LIN {X 0,Y 200.83,Z 502.645,A -85,B 0,C 180,E1 -22290.664,E2 -22290.664} C_VEL
LIN {X 0,Y 204.699,Z 493.667,A -85,B 0,C 180,E1 -22293.188,E2 -22293.188} C_VEL
LIN {X 0,Y 208.702,Z 483.459,A -85,B 0,C 180,E1 -22295.374,E2 -22295.374} C_VEL
LIN {X 0,Y 212.561,Z 471.698,A -85,B 0,C 180,E1 -22297.342,E2 -22297.342} C_VEL
LIN {X 0,Y 215.723,Z 459.835,A -85,B 0,C 180,E1 -22298.834,E2 -22298.834} C_VEL
LIN {X 0,Y 218.261,Z 447.534,A -85,B 0,C 180,E1 -22299.995,E2 -22299.995} C_VEL
LIN {X 0,Y 220.138,Z 434.92,A -85,B 0,C 180,E1 -22300.843,E2 -22300.843} C_VEL
LIN {X 0,Y 221.593,Z 419.626,A -85,B 0,C 180,E1 -22301.436,E2 -22301.436} C_VEL
LIN {X 0,Y 224.131,Z 384.01,A -85,B 0,C 180,E1 -22302.617,E2 -22302.617} C_VEL
LIN {X 0,Y 219.979,Z 374.841,A -85,B 0,C 180,E1 -22304.431,E2 -22304.431} C_VEL
LIN {X 0,Y 215.711,Z 367.271,A -85,B 0,C 180,E1 -22306.366,E2 -22306.366} C_VEL
LIN {X 0,Y 209.889,Z 358.051,A -85,B 0,C 180,E1 -22309.273,E2 -22309.273} C_VEL
LIN {X 0,Y 206.082,Z 352.787,A -85,B 0,C 180,E1 -22311.418,E2 -22311.418} C_VEL
LIN {X 0,Y 203.267,Z 348.749,A -85,B 0,C 180,E1 -22313.186,E2 -22313.186} C_VEL
LIN {X 0,Y 200.741,Z 345.417,A -85,B 0,C 180,E1 -22314.916,E2 -22314.916} C_VEL
LIN {X 0,Y 200.014,Z 344.287,A -85,B 0,C 180,E1 -22315.465,E2 -22315.465} C_VEL
LIN {X 0,Y 197.478,Z 341.831,A -85,B 0,C 180,E1 -22317.402,E2 -22317.402} C_VEL
LIN {X 0,Y 195.833,Z 338.802,A -85,B 0,C 180,E1 -22318.973,E2 -22318.973} C_VEL
LIN {X 0,Y 192.788,Z 336.052,A -85,B 0,C 180,E1 -22321.958,E2 -22321.958} C_VEL
LIN {X 0,Y 191.361,Z 333.353,A -85,B 0,C 180,E1 -22323.949,E2 -22323.949} C_VEL
LIN {X 0,Y 187.171,Z 330.783,A -85,B 0,C 180,E1 -22332.559,E2 -22332.559} C_VEL
LIN {X 0,Y 186.825,Z 330.456,A -85,B 0,C 180,E1 -22335.268,E2 -22335.268} C_VEL
LIN {X 0,Y 187.253,Z 331.063,A -85,B 0,C 180,E1 -22339.423,E2 -22339.423} C_VEL
LIN {X 0,Y 189.991,Z 333.324,A -85,B 0,C 180,E1 -22345.763,E2 -22345.763} C_VEL
LIN {X 0,Y 191.866,Z 335.584,A -85,B 0,C 180,E1 -22348.486,E2 -22348.486} C_VEL
LIN {X 0,Y 196.838,Z 342.088,A -85,B 0,C 180,E1 -22353.64,E2 -22353.64} C_VEL
LIN {X 0,Y 201.131,Z 348.366,A -85,B 0,C 180,E1 -22357.071,E2 -22357.071} C_VEL
LIN {X 0,Y 205.522,Z 355.246,A -85,B 0,C 180,E1 -22359.982,E2 -22359.982} C_VEL
LIN {X 0,Y 209.608,Z 362.229,A -85,B 0,C 180,E1 -22362.38,E2 -22362.38} C_VEL
LIN {X 0,Y 212.18,Z 366.87,A -85,B 0,C 180,E1 -22363.744,E2 -22363.744} C_VEL
LIN {X 0,Y 217.142,Z 376.724,A -85,B 0,C 180,E1 -22366.212,E2 -22366.212} C_VEL
LIN {X 0,Y 221.441,Z 387.148,A -85,B 0,C 180,E1 -22368.215,E2 -22368.215} C_VEL
LIN {X 0,Y 222.84,Z 391.134,A -85,B 0,C 180,E1 -22368.865,E2 -22368.865} C_VEL
LIN {X 0,Y 223.267,Z 398.392,A -85,B 0,C 180,E1 -22369.389,E2 -22369.389} C_VEL
LIN {X 0,Y 222.151,Z 414.024,A -85,B 0,C 180,E1 -22369.907,E2 -22369.907} C_VEL
LIN {X 0,Y 221.34,Z 419.86,A -85,B 0,C 180,E1 -22369.978,E2 -22369.978} C_VEL
LIN {X 0,Y 216.043,Z 438.883,A -85,B 0,C 180,E1 -22369.491,E2 -22369.491} C_VEL
LIN {X 0,Y 214.87,Z 444.674,A -85,B 0,C 180,E1 -22369.599,E2 -22369.599} C_VEL
LIN {X 0,Y 212.693,Z 457.533,A -85,B 0,C 180,E1 -22370.384,E2 -22370.384} C_VEL
LIN {X 0,Y 209.856,Z 469.525,A -85,B 0,C 180,E1 -22371.421,E2 -22371.421} C_VEL
LIN {X 0,Y 206.39,Z 481.375,A -85,B 0,C 180,E1 -22372.824,E2 -22372.824} C_VEL
LIN {X 0,Y 202.69,Z 492.094,A -85,B 0,C 180,E1 -22374.505,E2 -22374.505} C_VEL
LIN {X 0,Y 198.299,Z 502.866,A -85,B 0,C 180,E1 -22376.689,E2 -22376.689} C_VEL
LIN {X 0,Y 194.337,Z 511.664,A -85,B 0,C 180,E1 -22378.99,E2 -22378.99} C_VEL
LIN {X 0,Y 190.029,Z 520.315,A -85,B 0,C 180,E1 -22381.875,E2 -22381.875} C_VEL
LIN {X 0,Y 186.598,Z 526.823,A -85,B 0,C 180,E1 -22384.68,E2 -22384.68} C_VEL
LIN {X 0,Y 183.631,Z 532.054,A -85,B 0,C 180,E1 -22387.507,E2 -22387.507} C_VEL
LIN {X 0,Y 180.942,Z 536.694,A -85,B 0,C 180,E1 -22390.731,E2 -22390.731} C_VEL
LIN {X 0,Y 178.737,Z 540.277,A -85,B 0,C 180,E1 -22394.032,E2 -22394.032} C_VEL
LIN {X 0,Y 177.762,Z 542.118,A -85,B 0,C 180,E1 -22396.286,E2 -22396.286} C_VEL
LIN {X 0,Y 176.452,Z 544.563,A -85,B 0,C 180,E1 -22400.841,E2 -22400.841} C_VEL
LIN {X 0,Y 176.134,Z 545.21,A -85,B 0,C 180,E1 -22403.133,E2 -22403.133} C_VEL
LIN {X 0,Y 175.989,Z 545.399,A -85,B 0,C 180,E1 -22406.716,E2 -22406.716} C_VEL
LIN {X 0,Y 176.24,Z 544.71,A -85,B 0,C 180,E1 -22410.007,E2 -22410.007} C_VEL
LIN {X 0,Y 176.072,Z 542.876,A -85,B 0,C 180,E1 -22413.72,E2 -22413.72} C_VEL
LIN {X 0,Y 176.313,Z 539.323,A -85,B 0,C 180,E1 -22418.027,E2 -22418.027} C_VEL
LIN {X 0,Y 176.918,Z 535.242,A -85,B 0,C 180,E1 -22421.463,E2 -22421.463} C_VEL
LIN {X 0,Y 178.269,Z 528.927,A -85,B 0,C 180,E1 -22425.439,E2 -22425.439} C_VEL
LIN {X 0,Y 180.034,Z 522.023,A -85,B 0,C 180,E1 -22428.794,E2 -22428.794} C_VEL
LIN {X 0,Y 181.845,Z 515.368,A -85,B 0,C 180,E1 -22431.388,E2 -22431.388} C_VEL
LIN {X 0,Y 184.238,Z 506.448,A -85,B 0,C 180,E1 -22434.215,E2 -22434.215} C_VEL
LIN {X 0,Y 186.613,Z 497.088,A -85,B 0,C 180,E1 -22436.571,E2 -22436.571} C_VEL
LIN {X 0,Y 189.347,Z 485.491,A -85,B 0,C 180,E1 -22438.856,E2 -22438.856} C_VEL
LIN {X 0,Y 191.354,Z 475.884,A -85,B 0,C 180,E1 -22440.337,E2 -22440.337} C_VEL
LIN {X 0,Y 193.525,Z 463.742,A -85,B 0,C 180,E1 -22441.78,E2 -22441.78} C_VEL
LIN {X 0,Y 195.313,Z 450.462,A -85,B 0,C 180,E1 -22442.888,E2 -22442.888} C_VEL
LIN {X 0,Y 196.507,Z 437.019,A -85,B 0,C 180,E1 -22443.598,E2 -22443.598} C_VEL
LIN {X 0,Y 198.622,Z 393.171,A -85,B 0,C 180,E1 -22445.244,E2 -22445.244} C_VEL
LIN {X 0,Y 196.265,Z 372.863,A -85,B 0,C 180,E1 -22446.538,E2 -22446.538} C_VEL
LIN {X 0,Y 189.315,Z 354.681,A -85,B 0,C 180,E1 -22448.589,E2 -22448.589} C_VEL
LIN {X 0,Y 183.233,Z 340.766,A -85,B 0,C 180,E1 -22450.438,E2 -22450.438} C_VEL
LIN {X 0,Y 179.626,Z 333.029,A -85,B 0,C 180,E1 -22451.601,E2 -22451.601} C_VEL
LIN {X 0,Y 178.398,Z 328.269,A -85,B 0,C 180,E1 -22454.545,E2 -22454.545} C_VEL
LIN {X 0,Y 178.408,Z 328.261,A -85,B 0,C 180,E1 -22458.464,E2 -22458.464} C_VEL
LIN {X 0,Y 178.429,Z 328.26,A -85,B 0,C 180,E1 -22463.784,E2 -22463.784} C_VEL
LIN {X 0,Y 178.495,Z 328.252,A -85,B 0,C 180,E1 -22466.548,E2 -22466.548} C_VEL
LIN {X 0,Y 178.532,Z 328.242,A -85,B 0,C 180,E1 -22470.01,E2 -22470.01} C_VEL
LIN {X 0,Y 178.53,Z 328.241,A -85,B 0,C 180,E1 -22474.888,E2 -22474.888} C_VEL
LIN {X 0,Y 178.616,Z 328.213,A -85,B 0,C 180,E1 -22481.653,E2 -22481.653} C_VEL
LIN {X 0,Y 178.649,Z 328.216,A -85,B 0,C 180,E1 -22486.347,E2 -22486.347} C_VEL
LIN {X 0,Y 178.915,Z 328.199,A -85,B 0,C 180,E1 -22490.96,E2 -22490.96} C_VEL
LIN {X 0,Y 179.145,Z 328.121,A -85,B 0,C 180,E1 -22497.752,E2 -22497.752} C_VEL
LIN {X 0,Y 179.367,Z 328.106,A -85,B 0,C 180,E1 -22500,E2 -22500} C_VEL
LIN {X 0,Y 178.853,Z 328.204,A -85,B 0,C 180,E1 -22504.508,E2 -22504.508} C_VEL
LIN {X 0,Y 178.909,Z 328.191,A -85,B 0,C 180,E1 -22509.04,E2 -22509.04} C_VEL
LIN {X 0,Y 178.644,Z 328.231,A -85,B 0,C 180,E1 -22513.653,E2 -22513.653} C_VEL
LIN {X 0,Y 178.564,Z 328.226,A -85,B 0,C 180,E1 -22519.15,E2 -22519.15} C_VEL
LIN {X 0,Y 178.474,Z 328.248,A -85,B 0,C 180,E1 -22525.073,E2 -22525.073} C_VEL
LIN {X 0,Y 178.44,Z 328.213,A -85,B 0,C 180,E1 -22529.939,E2 -22529.939} C_VEL
LIN {X 0,Y 178.475,Z 328.226,A -85,B 0,C 180,E1 -22534.207,E2 -22534.207} C_VEL
LIN {X 0,Y 178.396,Z 328.262,A -85,B 0,C 180,E1 -22539.075,E2 -22539.075} C_VEL
LIN {X 0,Y 178.401,Z 328.255,A -85,B 0,C 180,E1 -22542.045,E2 -22542.045} C_VEL
LIN {X 0,Y 178.4,Z 328.262,A -85,B 0,C 180,E1 -22545.162,E2 -22545.162} C_VEL
LIN {X 0,Y 178.405,Z 328.257,A -85,B 0,C 180,E1 -22548.459,E2 -22548.459} C_VEL
LIN {X 0,Y 178.428,Z 328.259,A -85,B 0,C 180,E1 -22553.778,E2 -22553.778} C_VEL
LIN {X 0,Y 178.491,Z 328.248,A -85,B 0,C 180,E1 -22556.542,E2 -22556.542} C_VEL
LIN {X 0,Y 178.45,Z 328.256,A -85,B 0,C 180,E1 -22561.79,E2 -22561.79} C_VEL
LIN {X 0,Y 178.524,Z 328.251,A -85,B 0,C 180,E1 -22564.884,E2 -22564.884} C_VEL
LIN {X 0,Y 178.615,Z 328.239,A -85,B 0,C 180,E1 -22571.646,E2 -22571.646} C_VEL
LIN {X 0,Y 178.649,Z 328.233,A -85,B 0,C 180,E1 -22576.341,E2 -22576.341} C_VEL
LIN {X 0,Y 178.889,Z 328.197,A -85,B 0,C 180,E1 -22580.648,E2 -22580.648} C_VEL
LIN {X 0,Y 179.956,Z 331.094,A -85,B 0,C 180,E1 -22581.05,E2 -22581.05} C_VEL
LIN {X 0,Y 181.368,Z 333.406,A -85,B 0,C 180,E1 -22581.463,E2 -22581.463} C_VEL
LIN {X 0,Y 192.448,Z 353.773,A -85,B 0,C 180,E1 -22584.59,E2 -22584.59} C_VEL
LIN {X 0,Y 195.428,Z 360.834,A -85,B 0,C 180,E1 -22585.432,E2 -22585.432} C_VEL
LIN {X 0,Y 199.503,Z 371.756,A -85,B 0,C 180,E1 -22586.588,E2 -22586.588} C_VEL
LIN {X 0,Y 196.857,Z 422.474,A -85,B 0,C 180,E1 -22588.451,E2 -22588.451} C_VEL
LIN {X 0,Y 195.825,Z 436.185,A -85,B 0,C 180,E1 -22589.169,E2 -22589.169} C_VEL
LIN {X 0,Y 194.345,Z 449.201,A -85,B 0,C 180,E1 -22590.252,E2 -22590.252} C_VEL
LIN {X 0,Y 192.63,Z 460.504,A -85,B 0,C 180,E1 -22591.561,E2 -22591.561} C_VEL
LIN {X 0,Y 190.363,Z 472.121,A -85,B 0,C 180,E1 -22593.326,E2 -22593.326} C_VEL
LIN {X 0,Y 187.664,Z 483.863,A -85,B 0,C 180,E1 -22595.634,E2 -22595.634} C_VEL
LIN {X 0,Y 185.242,Z 493.538,A -85,B 0,C 180,E1 -22598.08,E2 -22598.08} C_VEL
LIN {X 0,Y 182.743,Z 502.914,A -85,B 0,C 180,E1 -22601.078,E2 -22601.078} C_VEL
LIN {X 0,Y 180.661,Z 510.535,A -85,B 0,C 180,E1 -22604.143,E2 -22604.143} C_VEL
LIN {X 0,Y 178.785,Z 517.533,A -85,B 0,C 180,E1 -22607.728,E2 -22607.728} C_VEL
LIN {X 0,Y 177.599,Z 522.314,A -85,B 0,C 180,E1 -22610.855,E2 -22610.855} C_VEL
LIN {X 0,Y 176.558,Z 526.913,A -85,B 0,C 180,E1 -22614.845,E2 -22614.845} C_VEL
LIN {X 0,Y 175.856,Z 529.978,A -85,B 0,C 180,E1 -22618.647,E2 -22618.647} C_VEL
LIN {X 0,Y 175.713,Z 532.023,A -85,B 0,C 180,E1 -22622.866,E2 -22622.866} C_VEL
LIN {X 0,Y 176.173,Z 532.682,A -85,B 0,C 180,E1 -22627.074,E2 -22627.074} C_VEL
LIN {X 0,Y 177.212,Z 532.051,A -85,B 0,C 180,E1 -22631.104,E2 -22631.104} C_VEL
LIN {X 0,Y 178.825,Z 530.233,A -85,B 0,C 180,E1 -22635.011,E2 -22635.011} C_VEL
LIN {X 0,Y 180.931,Z 527.349,A -85,B 0,C 180,E1 -22638.674,E2 -22638.674} C_VEL
LIN {X 0,Y 183.628,Z 523.283,A -85,B 0,C 180,E1 -22642.239,E2 -22642.239} C_VEL
LIN {X 0,Y 187.054,Z 517.798,A -85,B 0,C 180,E1 -22645.731,E2 -22645.731} C_VEL
LIN {X 0,Y 190.973,Z 510.931,A -85,B 0,C 180,E1 -22648.988,E2 -22648.988} C_VEL
LIN {X 0,Y 194.817,Z 503.511,A -85,B 0,C 180,E1 -22651.719,E2 -22651.719} C_VEL
LIN {X 0,Y 198.856,Z 494.672,A -85,B 0,C 180,E1 -22654.296,E2 -22654.296} C_VEL
LIN {X 0,Y 203.028,Z 484.688,A -85,B 0,C 180,E1 -22656.512,E2 -22656.512} C_VEL
LIN {X 0,Y 207.024,Z 473.241,A -85,B 0,C 180,E1 -22658.5,E2 -22658.5} C_VEL
LIN {X 0,Y 210.444,Z 461.357,A -85,B 0,C 180,E1 -22660.072,E2 -22660.072} C_VEL
LIN {X 0,Y 213.229,Z 448.861,A -85,B 0,C 180,E1 -22661.289,E2 -22661.289} C_VEL
LIN {X 0,Y 215.21,Z 436.521,A -85,B 0,C 180,E1 -22662.156,E2 -22662.156} C_VEL
LIN {X 0,Y 216.659,Z 423.215,A -85,B 0,C 180,E1 -22662.717,E2 -22662.717} C_VEL
LIN {X 0,Y 219.329,Z 386.42,A -85,B 0,C 180,E1 -22663.972,E2 -22663.972} C_VEL
LIN {X 0,Y 215.48,Z 378.059,A -85,B 0,C 180,E1 -22665.77,E2 -22665.77} C_VEL
LIN {X 0,Y 210.857,Z 369.986,A -85,B 0,C 180,E1 -22668.053,E2 -22668.053} C_VEL
LIN {X 0,Y 206.612,Z 363.273,A -85,B 0,C 180,E1 -22670.365,E2 -22670.365} C_VEL
LIN {X 0,Y 203.492,Z 358.724,A -85,B 0,C 180,E1 -22672.232,E2 -22672.232} C_VEL
LIN {X 0,Y 200.871,Z 354.901,A -85,B 0,C 180,E1 -22673.975,E2 -22673.975} C_VEL
LIN {X 0,Y 198.307,Z 351.201,A -85,B 0,C 180,E1 -22675.872,E2 -22675.872} C_VEL
LIN {X 0,Y 195.3,Z 347.833,A -85,B 0,C 180,E1 -22678.333,E2 -22678.333} C_VEL
LIN {X 0,Y 194.033,Z 345.46,A -85,B 0,C 180,E1 -22679.614,E2 -22679.614} C_VEL
LIN {X 0,Y 191.184,Z 342.587,A -85,B 0,C 180,E1 -22682.634,E2 -22682.634} C_VEL
LIN {X 0,Y 190.098,Z 340.349,A -85,B 0,C 180,E1 -22684.24,E2 -22684.24} C_VEL
LIN {X 0,Y 186.173,Z 337.836,A -85,B 0,C 180,E1 -22692.533,E2 -22692.533} C_VEL
LIN {X 0,Y 185.832,Z 337.475,A -85,B 0,C 180,E1 -22695.351,E2 -22695.351} C_VEL
LIN {X 0,Y 186.245,Z 338.113,A -85,B 0,C 180,E1 -22699.406,E2 -22699.406} C_VEL
LIN {X 0,Y 188.814,Z 340.289,A -85,B 0,C 180,E1 -22705.528,E2 -22705.528} C_VEL
LIN {X 0,Y 190.361,Z 342.23,A -85,B 0,C 180,E1 -22707.88,E2 -22707.88} C_VEL
LIN {X 0,Y 195.249,Z 349.146,A -85,B 0,C 180,E1 -22713.255,E2 -22713.255} C_VEL
LIN {X 0,Y 199.597,Z 355.746,A -85,B 0,C 180,E1 -22716.837,E2 -22716.837} C_VEL
LIN {X 0,Y 202.918,Z 361.212,A -85,B 0,C 180,E1 -22719.153,E2 -22719.153} C_VEL
LIN {X 0,Y 206.469,Z 367.403,A -85,B 0,C 180,E1 -22721.362,E2 -22721.362} C_VEL
LIN {X 0,Y 209.173,Z 372.611,A -85,B 0,C 180,E1 -22722.918,E2 -22722.918} C_VEL
LIN {X 0,Y 213.437,Z 381.344,A -85,B 0,C 180,E1 -22725.168,E2 -22725.168} C_VEL
LIN {X 0,Y 217.495,Z 391.631,A -85,B 0,C 180,E1 -22727.209,E2 -22727.209} C_VEL
LIN {X 0,Y 218.417,Z 394.335,A -85,B 0,C 180,E1 -22727.666,E2 -22727.666} C_VEL
LIN {X 0,Y 218.637,Z 399.043,A -85,B 0,C 180,E1 -22728.005,E2 -22728.005} C_VEL
LIN {X 0,Y 215.29,Z 441.072,A -85,B 0,C 180,E1 -22729.427,E2 -22729.427} C_VEL
LIN {X 0,Y 214.87,Z 444.674,A -85,B 0,C 180,E1 -22729.599,E2 -22729.599} C_VEL
LIN {X 0,Y 213.53,Z 450.424,A -85,B 0,C 180,E1 -22729.742,E2 -22729.742} C_VEL
LIN {X 0,Y 209.822,Z 459.643,A -85,B 0,C 180,E1 -22729.786,E2 -22729.786} C_VEL
LIN {X 0,Y 205.72,Z 468.593,A -85,B 0,C 180,E1 -22730.021,E2 -22730.021} C_VEL
LIN {X 0,Y 203.768,Z 473.909,A -85,B 0,C 180,E1 -22730.471,E2 -22730.471} C_VEL
LIN {X 0,Y 199.843,Z 485.685,A -85,B 0,C 180,E1 -22732.028,E2 -22732.028} C_VEL
LIN {X 0,Y 195.599,Z 496.635,A -85,B 0,C 180,E1 -22733.97,E2 -22733.97} C_VEL
LIN {X 0,Y 190.739,Z 507.337,A -85,B 0,C 180,E1 -22736.459,E2 -22736.459} C_VEL
LIN {X 0,Y 186.019,Z 516.738,A -85,B 0,C 180,E1 -22739.344,E2 -22739.344} C_VEL
LIN {X 0,Y 181.766,Z 524.321,A -85,B 0,C 180,E1 -22742.366,E2 -22742.366} C_VEL
LIN {X 0,Y 178.237,Z 530.459,A -85,B 0,C 180,E1 -22745.552,E2 -22745.552} C_VEL
LIN {X 0,Y 175.139,Z 535.376,A -85,B 0,C 180,E1 -22748.839,E2 -22748.839} C_VEL
LIN {X 0,Y 172.621,Z 539.202,A -85,B 0,C 180,E1 -22752.23,E2 -22752.23} C_VEL
LIN {X 0,Y 170.824,Z 542.038,A -85,B 0,C 180,E1 -22755.718,E2 -22755.718} C_VEL
LIN {X 0,Y 169.41,Z 544.396,A -85,B 0,C 180,E1 -22760.457,E2 -22760.457} C_VEL
LIN {X 0,Y 169.086,Z 544.994,A -85,B 0,C 180,E1 -22762.845,E2 -22762.845} C_VEL
LIN {X 0,Y 168.906,Z 545.055,A -85,B 0,C 180,E1 -22766.989,E2 -22766.989} C_VEL
LIN {X 0,Y 169.159,Z 544.341,A -85,B 0,C 180,E1 -22770.008,E2 -22770.008} C_VEL
LIN {X 0,Y 168.981,Z 542.671,A -85,B 0,C 180,E1 -22773.465,E2 -22773.465} C_VEL
LIN {X 0,Y 169.27,Z 538.737,A -85,B 0,C 180,E1 -22778.363,E2 -22778.363} C_VEL
LIN {X 0,Y 169.941,Z 534.558,A -85,B 0,C 180,E1 -22781.941,E2 -22781.941} C_VEL
LIN {X 0,Y 171.383,Z 528.135,A -85,B 0,C 180,E1 -22786.076,E2 -22786.076} C_VEL
LIN {X 0,Y 173.272,Z 521.111,A -85,B 0,C 180,E1 -22789.556,E2 -22789.556} C_VEL
LIN {X 0,Y 175.044,Z 514.752,A -85,B 0,C 180,E1 -22792.087,E2 -22792.087} C_VEL
LIN {X 0,Y 177.7,Z 505.18,A -85,B 0,C 180,E1 -22795.167,E2 -22795.167} C_VEL
LIN {X 0,Y 180.311,Z 495.627,A -85,B 0,C 180,E1 -22797.577,E2 -22797.577} C_VEL
LIN {X 0,Y 182.778,Z 485.195,A -85,B 0,C 180,E1 -22799.679,E2 -22799.679} C_VEL
LIN {X 0,Y 184.856,Z 475.582,A -85,B 0,C 180,E1 -22801.204,E2 -22801.204} C_VEL
LIN {X 0,Y 187.108,Z 463.441,A -85,B 0,C 180,E1 -22802.686,E2 -22802.686} C_VEL
LIN {X 0,Y 188.981,Z 449.999,A -85,B 0,C 180,E1 -22803.832,E2 -22803.832} C_VEL
LIN {X 0,Y 190.159,Z 436.642,A -85,B 0,C 180,E1 -22804.558,E2 -22804.558} C_VEL
LIN {X 0,Y 192.336,Z 393.741,A -85,B 0,C 180,E1 -22806.211,E2 -22806.211} C_VEL
LIN {X 0,Y 190.278,Z 375.38,A -85,B 0,C 180,E1 -22807.42,E2 -22807.42} C_VEL
LIN {X 0,Y 183.313,Z 356.878,A -85,B 0,C 180,E1 -22809.613,E2 -22809.613} C_VEL
LIN {X 0,Y 176.281,Z 341.004,A -85,B 0,C 180,E1 -22811.873,E2 -22811.873} C_VEL
LIN {X 0,Y 172.235,Z 332.782,A -85,B 0,C 180,E1 -22813.232,E2 -22813.232} C_VEL
LIN {X 0,Y 171.351,Z 329.145,A -85,B 0,C 180,E1 -22815.619,E2 -22815.619} C_VEL
LIN {X 0,Y 171.353,Z 329.141,A -85,B 0,C 180,E1 -22821.202,E2 -22821.202} C_VEL
LIN {X 0,Y 171.408,Z 329.131,A -85,B 0,C 180,E1 -22825.096,E2 -22825.096} C_VEL
LIN {X 0,Y 171.458,Z 329.125,A -85,B 0,C 180,E1 -22830.536,E2 -22830.536} C_VEL
LIN {X 0,Y 171.449,Z 329.125,A -85,B 0,C 180,E1 -22835.8,E2 -22835.8} C_VEL
LIN {X 0,Y 171.517,Z 329.103,A -85,B 0,C 180,E1 -22840.864,E2 -22840.864} C_VEL
LIN {X 0,Y 171.563,Z 329.089,A -85,B 0,C 180,E1 -22845.772,E2 -22845.772} C_VEL
LIN {X 0,Y 171.854,Z 329.077,A -85,B 0,C 180,E1 -22850.585,E2 -22850.585} C_VEL
LIN {X 0,Y 171.81,Z 329.052,A -85,B 0,C 180,E1 -22855.307,E2 -22855.307} C_VEL
LIN {X 0,Y 172.331,Z 328.981,A -85,B 0,C 180,E1 -22860,E2 -22860} C_VEL
LIN {X 0,Y 171.802,Z 329.082,A -85,B 0,C 180,E1 -22864.693,E2 -22864.693} C_VEL
LIN {X 0,Y 171.849,Z 329.067,A -85,B 0,C 180,E1 -22869.415,E2 -22869.415} C_VEL
LIN {X 0,Y 171.559,Z 329.114,A -85,B 0,C 180,E1 -22874.229,E2 -22874.229} C_VEL
LIN {X 0,Y 171.488,Z 329.108,A -85,B 0,C 180,E1 -22879.496,E2 -22879.496} C_VEL
LIN {X 0,Y 171.411,Z 329.127,A -85,B 0,C 180,E1 -22885.566,E2 -22885.566} C_VEL
LIN {X 0,Y 171.376,Z 329.086,A -85,B 0,C 180,E1 -22890.541,E2 -22890.541} C_VEL
LIN {X 0,Y 171.398,Z 329.114,A -85,B 0,C 180,E1 -22895.034,E2 -22895.034} C_VEL
LIN {X 0,Y 171.352,Z 329.141,A -85,B 0,C 180,E1 -22898.798,E2 -22898.798} C_VEL
LIN {X 0,Y 171.327,Z 329.138,A -85,B 0,C 180,E1 -22904.216,E2 -22904.216} C_VEL
LIN {X 0,Y 171.338,Z 329.134,A -85,B 0,C 180,E1 -22908.976,E2 -22908.976} C_VEL
LIN {X 0,Y 171.369,Z 329.139,A -85,B 0,C 180,E1 -22912.03,E2 -22912.03} C_VEL
LIN {X 0,Y 171.407,Z 329.128,A -85,B 0,C 180,E1 -22915.089,E2 -22915.089} C_VEL
LIN {X 0,Y 171.416,Z 329.132,A -85,B 0,C 180,E1 -22920.522,E2 -22920.522} C_VEL
LIN {X 0,Y 171.444,Z 329.128,A -85,B 0,C 180,E1 -22925.793,E2 -22925.793} C_VEL
LIN {X 0,Y 171.515,Z 329.12,A -85,B 0,C 180,E1 -22930.858,E2 -22930.858} C_VEL
LIN {X 0,Y 171.563,Z 329.116,A -85,B 0,C 180,E1 -22935.765,E2 -22935.765} C_VEL
LIN {X 0,Y 171.787,Z 329.153,A -85,B 0,C 180,E1 -22939.136,E2 -22939.136} C_VEL
LIN {X 0,Y 172.737,Z 331.778,A -85,B 0,C 180,E1 -22939.501,E2 -22939.501} C_VEL
LIN {X 0,Y 174.49,Z 334.545,A -85,B 0,C 180,E1 -22940.051,E2 -22940.051} C_VEL
LIN {X 0,Y 181.384,Z 346.939,A -85,B 0,C 180,E1 -22942.166,E2 -22942.166} C_VEL
LIN {X 0,Y 187.226,Z 357.999,A -85,B 0,C 180,E1 -22943.848,E2 -22943.848} C_VEL
LIN {X 0,Y 189.758,Z 364.031,A -85,B 0,C 180,E1 -22944.602,E2 -22944.602} C_VEL
LIN {X 0,Y 193.239,Z 373.45,A -85,B 0,C 180,E1 -22945.649,E2 -22945.649} C_VEL
LIN {X 0,Y 190.098,Z 429.382,A -85,B 0,C 180,E1 -22947.812,E2 -22947.812} C_VEL
LIN {X 0,Y 188.76,Z 443.002,A -85,B 0,C 180,E1 -22948.754,E2 -22948.754} C_VEL
LIN {X 0,Y 187.083,Z 455.192,A -85,B 0,C 180,E1 -22949.993,E2 -22949.993} C_VEL
LIN {X 0,Y 184.925,Z 467.034,A -85,B 0,C 180,E1 -22951.626,E2 -22951.626} C_VEL
LIN {X 0,Y 182.333,Z 478.517,A -85,B 0,C 180,E1 -22953.683,E2 -22953.683} C_VEL
LIN {X 0,Y 179.65,Z 489.272,A -85,B 0,C 180,E1 -22956.168,E2 -22956.168} C_VEL
LIN {X 0,Y 176.982,Z 499.215,A -85,B 0,C 180,E1 -22959.131,E2 -22959.131} C_VEL
LIN {X 0,Y 174.633,Z 507.378,A -85,B 0,C 180,E1 -22962.189,E2 -22962.189} C_VEL
LIN {X 0,Y 172.78,Z 514.053,A -85,B 0,C 180,E1 -22965.322,E2 -22965.322} C_VEL
LIN {X 0,Y 171.047,Z 520.492,A -85,B 0,C 180,E1 -22969.181,E2 -22969.181} C_VEL
LIN {X 0,Y 169.896,Z 525.338,A -85,B 0,C 180,E1 -22973.02,E2 -22973.02} C_VEL
LIN {X 0,Y 168.936,Z 529.177,A -85,B 0,C 180,E1 -22977.223,E2 -22977.223} C_VEL
LIN {X 0,Y 168.632,Z 530.945,A -85,B 0,C 180,E1 -22979.996,E2 -22979.996} C_VEL
LIN {X 0,Y 168.658,Z 532.399,A -85,B 0,C 180,E1 -22983.55,E2 -22983.55} C_VEL
LIN {X 0,Y 169.214,Z 532.944,A -85,B 0,C 180,E1 -22987.895,E2 -22987.895} C_VEL
LIN {X 0,Y 170.456,Z 532.233,A -85,B 0,C 180,E1 -22992.085,E2 -22992.085} C_VEL
LIN {X 0,Y 172.19,Z 530.389,A -85,B 0,C 180,E1 -22996.063,E2 -22996.063} C_VEL
LIN {X 0,Y 174.548,Z 527.417,A -85,B 0,C 180,E1 -22999.892,E2 -22999.892} C_VEL
LIN {X 0,Y 177.523,Z 523.262,A -85,B 0,C 180,E1 -23003.57,E2 -23003.57} C_VEL
LIN {X 0,Y 181.152,Z 517.746,A -85,B 0,C 180,E1 -23007.102,E2 -23007.102} C_VEL
LIN {X 0,Y 185.558,Z 510.459,A -85,B 0,C 180,E1 -23010.568,E2 -23010.568} C_VEL
LIN {X 0,Y 189.193,Z 503.804,A -85,B 0,C 180,E1 -23013.043,E2 -23013.043} C_VEL
LIN {X 0,Y 193.096,Z 495.737,A -85,B 0,C 180,E1 -23015.468,E2 -23015.468} C_VEL
LIN {X 0,Y 197.445,Z 486.043,A -85,B 0,C 180,E1 -23017.711,E2 -23017.711} C_VEL
LIN {X 0,Y 201.667,Z 474.702,A -85,B 0,C 180,E1 -23019.741,E2 -23019.741} C_VEL
LIN {X 0,Y 205.307,Z 462.812,A -85,B 0,C 180,E1 -23021.372,E2 -23021.372} C_VEL
LIN {X 0,Y 208.172,Z 451.075,A -85,B 0,C 180,E1 -23022.562,E2 -23022.562} C_VEL
LIN {X 0,Y 210.349,Z 438.62,A -85,B 0,C 180,E1 -23023.489,E2 -23023.489} C_VEL
LIN {X 0,Y 211.912,Z 425.974,A -85,B 0,C 180,E1 -23024.071,E2 -23024.071} C_VEL
LIN {X 0,Y 214.738,Z 389.202,A -85,B 0,C 180,E1 -23025.344,E2 -23025.344} C_VEL
LIN {X 0,Y 211.148,Z 381.471,A -85,B 0,C 180,E1 -23027.17,E2 -23027.17} C_VEL
LIN {X 0,Y 206.112,Z 372.587,A -85,B 0,C 180,E1 -23029.896,E2 -23029.896} C_VEL
LIN {X 0,Y 201.292,Z 365.158,A -85,B 0,C 180,E1 -23032.844,E2 -23032.844} C_VEL
LIN {X 0,Y 198.609,Z 361.116,A -85,B 0,C 180,E1 -23034.742,E2 -23034.742} C_VEL
LIN {X 0,Y 195.812,Z 357.15,A -85,B 0,C 180,E1 -23036.925,E2 -23036.925} C_VEL
LIN {X 0,Y 193.168,Z 353.8,A -85,B 0,C 180,E1 -23039.303,E2 -23039.303} C_VEL
LIN {X 0,Y 192.278,Z 352.093,A -85,B 0,C 180,E1 -23040.262,E2 -23040.262} C_VEL
LIN {X 0,Y 189.607,Z 349.122,A -85,B 0,C 180,E1 -23043.32,E2 -23043.32} C_VEL
LIN {X 0,Y 188.649,Z 347.23,A -85,B 0,C 180,E1 -23044.802,E2 -23044.802} C_VEL
LIN {X 0,Y 185.158,Z 344.863,A -85,B 0,C 180,E1 -23052.603,E2 -23052.603} C_VEL
LIN {X 0,Y 184.837,Z 344.512,A -85,B 0,C 180,E1 -23055.436,E2 -23055.436} C_VEL
LIN {X 0,Y 185.225,Z 345.138,A -85,B 0,C 180,E1 -23059.323,E2 -23059.323} C_VEL
LIN {X 0,Y 187.545,Z 347.156,A -85,B 0,C 180,E1 -23065.129,E2 -23065.129} C_VEL
LIN {X 0,Y 189.002,Z 349.142,A -85,B 0,C 180,E1 -23067.461,E2 -23067.461} C_VEL
LIN {X 0,Y 193.416,Z 355.655,A -85,B 0,C 180,E1 -23072.599,E2 -23072.599} C_VEL
LIN {X 0,Y 197.298,Z 361.813,A -85,B 0,C 180,E1 -23075.997,E2 -23075.997} C_VEL
LIN {X 0,Y 200.497,Z 367.393,A -85,B 0,C 180,E1 -23078.392,E2 -23078.392} C_VEL
LIN {X 0,Y 203.661,Z 373.141,A -85,B 0,C 180,E1 -23080.474,E2 -23080.474} C_VEL
LIN {X 0,Y 206.909,Z 379.671,A -85,B 0,C 180,E1 -23082.462,E2 -23082.462} C_VEL
LIN {X 0,Y 210.367,Z 387.384,A -85,B 0,C 180,E1 -23084.393,E2 -23084.393} C_VEL
LIN {X 0,Y 213.974,Z 397.134,A -85,B 0,C 180,E1 -23086.356,E2 -23086.356} C_VEL
LIN {X 0,Y 214.041,Z 400.802,A -85,B 0,C 180,E1 -23086.6,E2 -23086.6} C_VEL
LIN {X 0,Y 210.663,Z 441.246,A -85,B 0,C 180,E1 -23087.984,E2 -23087.984} C_VEL
LIN {X 0,Y 208.483,Z 454.951,A -85,B 0,C 180,E1 -23088.753,E2 -23088.753} C_VEL
LIN {X 0,Y 205.496,Z 467.74,A -85,B 0,C 180,E1 -23089.807,E2 -23089.807} C_VEL
LIN {X 0,Y 203.768,Z 473.909,A -85,B 0,C 180,E1 -23090.471,E2 -23090.471} C_VEL
LIN {X 0,Y 201.664,Z 479.204,A -85,B 0,C 180,E1 -23090.981,E2 -23090.981} C_VEL
LIN {X 0,Y 196.671,Z 487.503,A -85,B 0,C 180,E1 -23091.583,E2 -23091.583} C_VEL
LIN {X 0,Y 191.423,Z 495.415,A -85,B 0,C 180,E1 -23092.389,E2 -23092.389} C_VEL
LIN {X 0,Y 188.949,Z 499.962,A -85,B 0,C 180,E1 -23093.225,E2 -23093.225} C_VEL
LIN {X 0,Y 184.904,Z 508.147,A -85,B 0,C 180,E1 -23095.252,E2 -23095.252} C_VEL
LIN {X 0,Y 179.982,Z 517.29,A -85,B 0,C 180,E1 -23098.198,E2 -23098.198} C_VEL
LIN {X 0,Y 175.527,Z 524.704,A -85,B 0,C 180,E1 -23101.294,E2 -23101.294} C_VEL
LIN {X 0,Y 171.809,Z 530.698,A -85,B 0,C 180,E1 -23104.574,E2 -23104.574} C_VEL
LIN {X 0,Y 168.51,Z 535.505,A -85,B 0,C 180,E1 -23107.963,E2 -23107.963} C_VEL
LIN {X 0,Y 165.864,Z 539.231,A -85,B 0,C 180,E1 -23111.48,E2 -23111.48} C_VEL
LIN {X 0,Y 163.908,Z 541.973,A -85,B 0,C 180,E1 -23115.101,E2 -23115.101} C_VEL
LIN {X 0,Y 162.391,Z 544.235,A -85,B 0,C 180,E1 -23120.04,E2 -23120.04} C_VEL
LIN {X 0,Y 162.011,Z 544.75,A -85,B 0,C 180,E1 -23122.531,E2 -23122.531} C_VEL
LIN {X 0,Y 161.832,Z 544.663,A -85,B 0,C 180,E1 -23127.24,E2 -23127.24} C_VEL
LIN {X 0,Y 162.06,Z 543.972,A -85,B 0,C 180,E1 -23130.008,E2 -23130.008} C_VEL
LIN {X 0,Y 161.89,Z 542.484,A -85,B 0,C 180,E1 -23133.155,E2 -23133.155} C_VEL
LIN {X 0,Y 162.074,Z 539.326,A -85,B 0,C 180,E1 -23137.482,E2 -23137.482} C_VEL
LIN {X 0,Y 162.671,Z 535.433,A -85,B 0,C 180,E1 -23141.218,E2 -23141.218} C_VEL
LIN {X 0,Y 163.718,Z 530.357,A -85,B 0,C 180,E1 -23144.933,E2 -23144.933} C_VEL
LIN {X 0,Y 165.519,Z 523.962,A -85,B 0,C 180,E1 -23148.576,E2 -23148.576} C_VEL
LIN {X 0,Y 167.851,Z 515.905,A -85,B 0,C 180,E1 -23152.144,E2 -23152.144} C_VEL
LIN {X 0,Y 169.711,Z 509.48,A -85,B 0,C 180,E1 -23154.47,E2 -23154.47} C_VEL
LIN {X 0,Y 172.412,Z 499.791,A -85,B 0,C 180,E1 -23157.302,E2 -23157.302} C_VEL
LIN {X 0,Y 175.242,Z 489.062,A -85,B 0,C 180,E1 -23159.761,E2 -23159.761} C_VEL
LIN {X 0,Y 177.773,Z 478.751,A -85,B 0,C 180,E1 -23161.595,E2 -23161.595} C_VEL
LIN {X 0,Y 179.981,Z 467.562,A -85,B 0,C 180,E1 -23163.146,E2 -23163.146} C_VEL
LIN {X 0,Y 182.047,Z 454.416,A -85,B 0,C 180,E1 -23164.465,E2 -23164.465} C_VEL
LIN {X 0,Y 183.506,Z 441.468,A -85,B 0,C 180,E1 -23165.334,E2 -23165.334} C_VEL
LIN {X 0,Y 186.118,Z 395.461,A -85,B 0,C 180,E1 -23167.175,E2 -23167.175} C_VEL
LIN {X 0,Y 184.344,Z 377.817,A -85,B 0,C 180,E1 -23168.364,E2 -23168.364} C_VEL
LIN {X 0,Y 177.367,Z 359.189,A -85,B 0,C 180,E1 -23170.674,E2 -23170.674} C_VEL
LIN {X 0,Y 170.502,Z 343.799,A -85,B 0,C 180,E1 -23173.01,E2 -23173.01} C_VEL
LIN {X 0,Y 164.867,Z 332.361,A -85,B 0,C 180,E1 -23175.088,E2 -23175.088} C_VEL
LIN {X 0,Y 164.271,Z 330.026,A -85,B 0,C 180,E1 -23176.802,E2 -23176.802} C_VEL
LIN {X 0,Y 164.3,Z 330.02,A -85,B 0,C 180,E1 -23180.358,E2 -23180.358} C_VEL
LIN {X 0,Y 164.336,Z 330.015,A -85,B 0,C 180,E1 -23186.223,E2 -23186.223} C_VEL
LIN {X 0,Y 164.399,Z 330.003,A -85,B 0,C 180,E1 -23189.136,E2 -23189.136} C_VEL
LIN {X 0,Y 164.415,Z 329.998,A -85,B 0,C 180,E1 -23194.694,E2 -23194.694} C_VEL
LIN {X 0,Y 164.427,Z 329.993,A -85,B 0,C 180,E1 -23200.119,E2 -23200.119} C_VEL
LIN {X 0,Y 164.491,Z 329.963,A -85,B 0,C 180,E1 -23205.146,E2 -23205.146} C_VEL
LIN {X 0,Y 164.775,Z 329.959,A -85,B 0,C 180,E1 -23210.177,E2 -23210.177} C_VEL
LIN {X 0,Y 164.834,Z 329.945,A -85,B 0,C 180,E1 -23212.651,E2 -23212.651} C_VEL
LIN {X 0,Y 165.294,Z 329.855,A -85,B 0,C 180,E1 -23220,E2 -23220} C_VEL
LIN {X 0,Y 164.751,Z 329.961,A -85,B 0,C 180,E1 -23224.894,E2 -23224.894} C_VEL
LIN {X 0,Y 164.826,Z 329.952,A -85,B 0,C 180,E1 -23227.349,E2 -23227.349} C_VEL
LIN {X 0,Y 164.711,Z 329.954,A -85,B 0,C 180,E1 -23231.054,E2 -23231.054} C_VEL
LIN {X 0,Y 164.443,Z 329.992,A -85,B 0,C 180,E1 -23237.408,E2 -23237.408} C_VEL
LIN {X 0,Y 164.43,Z 329.989,A -85,B 0,C 180,E1 -23239.995,E2 -23239.995} C_VEL
LIN {X 0,Y 164.344,Z 330.002,A -85,B 0,C 180,E1 -23246.088,E2 -23246.088} C_VEL
LIN {X 0,Y 164.315,Z 329.962,A -85,B 0,C 180,E1 -23251.184,E2 -23251.184} C_VEL
LIN {X 0,Y 164.333,Z 330,A -85,B 0,C 180,E1 -23255.644,E2 -23255.644} C_VEL
LIN {X 0,Y 164.295,Z 330.019,A -85,B 0,C 180,E1 -23259.915,E2 -23259.915} C_VEL
LIN {X 0,Y 164.291,Z 330.011,A -85,B 0,C 180,E1 -23263.339,E2 -23263.339} C_VEL
LIN {X 0,Y 164.269,Z 330.023,A -85,B 0,C 180,E1 -23266.794,E2 -23266.794} C_VEL
LIN {X 0,Y 164.298,Z 330.012,A -85,B 0,C 180,E1 -23270.351,E2 -23270.351} C_VEL
LIN {X 0,Y 164.335,Z 330.013,A -85,B 0,C 180,E1 -23274.347,E2 -23274.347} C_VEL
LIN {X 0,Y 164.378,Z 330.013,A -85,B 0,C 180,E1 -23279.125,E2 -23279.125} C_VEL
LIN {X 0,Y 164.402,Z 330.011,A -85,B 0,C 180,E1 -23284.685,E2 -23284.685} C_VEL
LIN {X 0,Y 164.424,Z 330.005,A -85,B 0,C 180,E1 -23290.111,E2 -23290.111} C_VEL
LIN {X 0,Y 164.491,Z 329.994,A -85,B 0,C 180,E1 -23295.139,E2 -23295.139} C_VEL
LIN {X 0,Y 164.609,Z 330.116,A -85,B 0,C 180,E1 -23297.432,E2 -23297.432} C_VEL
LIN {X 0,Y 165.72,Z 332.992,A -85,B 0,C 180,E1 -23297.881,E2 -23297.881} C_VEL
LIN {X 0,Y 167.275,Z 335.081,A -85,B 0,C 180,E1 -23298.388,E2 -23298.388} C_VEL
LIN {X 0,Y 173.112,Z 345.253,A -85,B 0,C 180,E1 -23300.331,E2 -23300.331} C_VEL
LIN {X 0,Y 181.862,Z 361.772,A -85,B 0,C 180,E1 -23303.017,E2 -23303.017} C_VEL
LIN {X 0,Y 184.419,Z 368.128,A -85,B 0,C 180,E1 -23303.823,E2 -23303.823} C_VEL
LIN {X 0,Y 187.085,Z 375.458,A -85,B 0,C 180,E1 -23304.675,E2 -23304.675} C_VEL
LIN {X 0,Y 183.836,Z 429.507,A -85,B 0,C 180,E1 -23306.806,E2 -23306.806} C_VEL
LIN {X 0,Y 182.414,Z 443.327,A -85,B 0,C 180,E1 -23307.785,E2 -23307.785} C_VEL
LIN {X 0,Y 180.531,Z 456.272,A -85,B 0,C 180,E1 -23309.156,E2 -23309.156} C_VEL
LIN {X 0,Y 178.277,Z 467.947,A -85,B 0,C 180,E1 -23310.84,E2 -23310.84} C_VEL
LIN {X 0,Y 175.586,Z 479.465,A -85,B 0,C 180,E1 -23312.997,E2 -23312.997} C_VEL
LIN {X 0,Y 172.842,Z 489.932,A -85,B 0,C 180,E1 -23315.534,E2 -23315.534} C_VEL
LIN {X 0,Y 169.943,Z 500.267,A -85,B 0,C 180,E1 -23318.763,E2 -23318.763} C_VEL
LIN {X 0,Y 167.462,Z 508.649,A -85,B 0,C 180,E1 -23322.104,E2 -23322.104} C_VEL
LIN {X 0,Y 165.233,Z 516.276,A -85,B 0,C 180,E1 -23326.04,E2 -23326.04} C_VEL
LIN {X 0,Y 163.595,Z 522.312,A -85,B 0,C 180,E1 -23330.091,E2 -23330.091} C_VEL
LIN {X 0,Y 162.379,Z 527.27,A -85,B 0,C 180,E1 -23334.644,E2 -23334.644} C_VEL
LIN {X 0,Y 161.693,Z 530.253,A -85,B 0,C 180,E1 -23338.551,E2 -23338.551} C_VEL
LIN {X 0,Y 161.508,Z 531.798,A -85,B 0,C 180,E1 -23341.466,E2 -23341.466} C_VEL
LIN {X 0,Y 161.627,Z 532.77,A -85,B 0,C 180,E1 -23344.409,E2 -23344.409} C_VEL
LIN {X 0,Y 162.351,Z 533.205,A -85,B 0,C 180,E1 -23348.812,E2 -23348.812} C_VEL
LIN {X 0,Y 163.806,Z 532.368,A -85,B 0,C 180,E1 -23353.336,E2 -23353.336} C_VEL
LIN {X 0,Y 165.638,Z 530.528,A -85,B 0,C 180,E1 -23357.244,E2 -23357.244} C_VEL
LIN {X 0,Y 168.234,Z 527.491,A -85,B 0,C 180,E1 -23361.198,E2 -23361.198} C_VEL
LIN {X 0,Y 171.514,Z 523.205,A -85,B 0,C 180,E1 -23365.018,E2 -23365.018} C_VEL
LIN {X 0,Y 175.462,Z 517.616,A -85,B 0,C 180,E1 -23368.62,E2 -23368.62} C_VEL
LIN {X 0,Y 180.029,Z 510.481,A -85,B 0,C 180,E1 -23372.066,E2 -23372.066} C_VEL
LIN {X 0,Y 184.245,Z 503.172,A -85,B 0,C 180,E1 -23374.777,E2 -23374.777} C_VEL
LIN {X 0,Y 188.545,Z 494.686,A -85,B 0,C 180,E1 -23377.275,E2 -23377.275} C_VEL
LIN {X 0,Y 192.755,Z 485.428,A -85,B 0,C 180,E1 -23379.378,E2 -23379.378} C_VEL
LIN {X 0,Y 197.222,Z 473.806,A -85,B 0,C 180,E1 -23381.428,E2 -23381.428} C_VEL
LIN {X 0,Y 200.757,Z 462.704,A -85,B 0,C 180,E1 -23382.93,E2 -23382.93} C_VEL
LIN {X 0,Y 203.799,Z 450.501,A -85,B 0,C 180,E1 -23384.16,E2 -23384.16} C_VEL
LIN {X 0,Y 206.032,Z 438.044,A -85,B 0,C 180,E1 -23385.075,E2 -23385.075} C_VEL
LIN {X 0,Y 207.69,Z 424.736,A -85,B 0,C 180,E1 -23385.66,E2 -23385.66} C_VEL
LIN {X 0,Y 210.331,Z 392.08,A -85,B 0,C 180,E1 -23386.785,E2 -23386.785} C_VEL
LIN {X 0,Y 206.796,Z 384.634,A -85,B 0,C 180,E1 -23388.708,E2 -23388.708} C_VEL
LIN {X 0,Y 201.623,Z 375.515,A -85,B 0,C 180,E1 -23391.818,E2 -23391.818} C_VEL
LIN {X 0,Y 196.699,Z 367.688,A -85,B 0,C 180,E1 -23395.293,E2 -23395.293} C_VEL
LIN {X 0,Y 193.691,Z 363.436,A -85,B 0,C 180,E1 -23397.766,E2 -23397.766} C_VEL
LIN {X 0,Y 191.131,Z 359.807,A -85,B 0,C 180,E1 -23400.263,E2 -23400.263} C_VEL
LIN {X 0,Y 190.42,Z 358.578,A -85,B 0,C 180,E1 -23401.057,E2 -23401.057} C_VEL
LIN {X 0,Y 187.976,Z 355.485,A -85,B 0,C 180,E1 -23404.145,E2 -23404.145} C_VEL
LIN {X 0,Y 187.294,Z 354.112,A -85,B 0,C 180,E1 -23405.268,E2 -23405.268} C_VEL
LIN {X 0,Y 184.145,Z 351.89,A -85,B 0,C 180,E1 -23412.673,E2 -23412.673} C_VEL
LIN {X 0,Y 183.934,Z 351.653,A -85,B 0,C 180,E1 -23417.246,E2 -23417.246} C_VEL
LIN {X 0,Y 186.186,Z 353.87,A -85,B 0,C 180,E1 -23424.533,E2 -23424.533} C_VEL
LIN {X 0,Y 187.581,Z 355.857,A -85,B 0,C 180,E1 -23426.91,E2 -23426.91} C_VEL
LIN {X 0,Y 191.505,Z 361.973,A -85,B 0,C 180,E1 -23431.806,E2 -23431.806} C_VEL
LIN {X 0,Y 195.033,Z 367.895,A -85,B 0,C 180,E1 -23435.134,E2 -23435.134} C_VEL
LIN {X 0,Y 197.964,Z 373.184,A -85,B 0,C 180,E1 -23437.47,E2 -23437.47} C_VEL
LIN {X 0,Y 201.892,Z 380.691,A -85,B 0,C 180,E1 -23440.205,E2 -23440.205} C_VEL
LIN {X 0,Y 206.367,Z 390.825,A -85,B 0,C 180,E1 -23443.018,E2 -23443.018} C_VEL
LIN {X 0,Y 209.758,Z 400.253,A -85,B 0,C 180,E1 -23445.004,E2 -23445.004} C_VEL
LIN {X 0,Y 206.569,Z 438.648,A -85,B 0,C 180,E1 -23446.346,E2 -23446.346} C_VEL
LIN {X 0,Y 204.561,Z 451.822,A -85,B 0,C 180,E1 -23447.031,E2 -23447.031} C_VEL
LIN {X 0,Y 201.618,Z 464.841,A -85,B 0,C 180,E1 -23448.035,E2 -23448.035} C_VEL
LIN {X 0,Y 198.057,Z 476.85,A -85,B 0,C 180,E1 -23449.317,E2 -23449.317} C_VEL
LIN {X 0,Y 193.884,Z 488.321,A -85,B 0,C 180,E1 -23450.975,E2 -23450.975} C_VEL
LIN {X 0,Y 189.039,Z 499.76,A -85,B 0,C 180,E1 -23453.178,E2 -23453.178} C_VEL
LIN {X 0,Y 188.949,Z 499.962,A -85,B 0,C 180,E1 -23453.225,E2 -23453.225} C_VEL
LIN {X 0,Y 186.427,Z 504.374,A -85,B 0,C 180,E1 -23454.149,E2 -23454.149} C_VEL
LIN {X 0,Y 178.204,Z 513.884,A -85,B 0,C 180,E1 -23456.037,E2 -23456.037} C_VEL
LIN {X 0,Y 173.7,Z 518.811,A -85,B 0,C 180,E1 -23457.408,E2 -23457.408} C_VEL
LIN {X 0,Y 171.966,Z 521.101,A -85,B 0,C 180,E1 -23458.287,E2 -23458.287} C_VEL
LIN {X 0,Y 167.948,Z 527.204,A -85,B 0,C 180,E1 -23461.247,E2 -23461.247} C_VEL
LIN {X 0,Y 164.175,Z 532.65,A -85,B 0,C 180,E1 -23464.665,E2 -23464.665} C_VEL
LIN {X 0,Y 160.964,Z 536.959,A -85,B 0,C 180,E1 -23468.225,E2 -23468.225} C_VEL
LIN {X 0,Y 158.317,Z 540.242,A -85,B 0,C 180,E1 -23471.906,E2 -23471.906} C_VEL
LIN {X 0,Y 156.065,Z 543.187,A -85,B 0,C 180,E1 -23476.997,E2 -23476.997} C_VEL
LIN {X 0,Y 155.392,Z 544.045,A -85,B 0,C 180,E1 -23479.587,E2 -23479.587} C_VEL
LIN {X 0,Y 154.756,Z 544.583,A -85,B 0,C 180,E1 -23484.798,E2 -23484.798} C_VEL
LIN {X 0,Y 154.775,Z 544.282,A -85,B 0,C 180,E1 -23487.406,E2 -23487.406} C_VEL
LIN {X 0,Y 154.964,Z 543.578,A -85,B 0,C 180,E1 -23490.008,E2 -23490.008} C_VEL
LIN {X 0,Y 154.815,Z 542.238,A -85,B 0,C 180,E1 -23492.903,E2 -23492.903} C_VEL
LIN {X 0,Y 154.893,Z 539.841,A -85,B 0,C 180,E1 -23496.521,E2 -23496.521} C_VEL
LIN {X 0,Y 155.405,Z 536.224,A -85,B 0,C 180,E1 -23500.43,E2 -23500.43} C_VEL
LIN {X 0,Y 156.381,Z 531.444,A -85,B 0,C 180,E1 -23504.318,E2 -23504.318} C_VEL
LIN {X 0,Y 158.399,Z 524.241,A -85,B 0,C 180,E1 -23508.772,E2 -23508.772} C_VEL
LIN {X 0,Y 160.823,Z 516.357,A -85,B 0,C 180,E1 -23512.488,E2 -23512.488} C_VEL
LIN {X 0,Y 162.327,Z 511.12,A -85,B 0,C 180,E1 -23514.521,E2 -23514.521} C_VEL
LIN {X 0,Y 165.083,Z 501.581,A -85,B 0,C 180,E1 -23517.586,E2 -23517.586} C_VEL
LIN {X 0,Y 167.698,Z 492.606,A -85,B 0,C 180,E1 -23519.852,E2 -23519.852} C_VEL
LIN {X 0,Y 170.585,Z 481.573,A -85,B 0,C 180,E1 -23522.042,E2 -23522.042} C_VEL
LIN {X 0,Y 172.824,Z 471.206,A -85,B 0,C 180,E1 -23523.653,E2 -23523.653} C_VEL
LIN {X 0,Y 175.085,Z 458.955,A -85,B 0,C 180,E1 -23525.072,E2 -23525.072} C_VEL
LIN {X 0,Y 176.775,Z 446.563,A -85,B 0,C 180,E1 -23526.085,E2 -23526.085} C_VEL
LIN {X 0,Y 177.914,Z 431.59,A -85,B 0,C 180,E1 -23526.837,E2 -23526.837} C_VEL
LIN {X 0,Y 179.969,Z 395.667,A -85,B 0,C 180,E1 -23528.284,E2 -23528.284} C_VEL
LIN {X 0,Y 178.367,Z 380.062,A -85,B 0,C 180,E1 -23529.385,E2 -23529.385} C_VEL
LIN {X 0,Y 171.698,Z 362.171,A -85,B 0,C 180,E1 -23531.713,E2 -23531.713} C_VEL
LIN {X 0,Y 165.428,Z 347.883,A -85,B 0,C 180,E1 -23533.981,E2 -23533.981} C_VEL
LIN {X 0,Y 159.244,Z 335.775,A -85,B 0,C 180,E1 -23536.292,E2 -23536.292} C_VEL
LIN {X 0,Y 157.481,Z 332.145,A -85,B 0,C 180,E1 -23537.016,E2 -23537.016} C_VEL
LIN {X 0,Y 157.18,Z 330.906,A -85,B 0,C 180,E1 -23537.992,E2 -23537.992} C_VEL
LIN {X 0,Y 157.269,Z 330.897,A -85,B 0,C 180,E1 -23543.559,E2 -23543.559} C_VEL
LIN {X 0,Y 157.303,Z 330.894,A -85,B 0,C 180,E1 -23548.1,E2 -23548.1} C_VEL
LIN {X 0,Y 157.325,Z 330.886,A -85,B 0,C 180,E1 -23553.467,E2 -23553.467} C_VEL
LIN {X 0,Y 157.371,Z 330.875,A -85,B 0,C 180,E1 -23559.704,E2 -23559.704} C_VEL
LIN {X 0,Y 157.423,Z 330.837,A -85,B 0,C 180,E1 -23564.463,E2 -23564.463} C_VEL
LIN {X 0,Y 157.698,Z 330.841,A -85,B 0,C 180,E1 -23569.731,E2 -23569.731} C_VEL
LIN {X 0,Y 157.772,Z 330.827,A -85,B 0,C 180,E1 -23572.32,E2 -23572.32} C_VEL
LIN {X 0,Y 158.256,Z 330.73,A -85,B 0,C 180,E1 -23580,E2 -23580} C_VEL
LIN {X 0,Y 157.764,Z 330.829,A -85,B 0,C 180,E1 -23587.68,E2 -23587.68} C_VEL
LIN {X 0,Y 157.64,Z 330.835,A -85,B 0,C 180,E1 -23591.219,E2 -23591.219} C_VEL
LIN {X 0,Y 157.421,Z 330.876,A -85,B 0,C 180,E1 -23595.538,E2 -23595.538} C_VEL
LIN {X 0,Y 157.314,Z 330.883,A -85,B 0,C 180,E1 -23600.941,E2 -23600.941} C_VEL
LIN {X 0,Y 157.278,Z 330.879,A -85,B 0,C 180,E1 -23606.647,E2 -23606.647} C_VEL
LIN {X 0,Y 157.251,Z 330.843,A -85,B 0,C 180,E1 -23612.433,E2 -23612.433} C_VEL
LIN {X 0,Y 157.267,Z 330.884,A -85,B 0,C 180,E1 -23616.44,E2 -23616.44} C_VEL
LIN {X 0,Y 157.198,Z 330.894,A -85,B 0,C 180,E1 -23622.115,E2 -23622.115} C_VEL
LIN {X 0,Y 157.198,Z 330.901,A -85,B 0,C 180,E1 -23627.878,E2 -23627.878} C_VEL
LIN {X 0,Y 157.268,Z 330.895,A -85,B 0,C 180,E1 -23633.551,E2 -23633.551} C_VEL
LIN {X 0,Y 157.292,Z 330.895,A -85,B 0,C 180,E1 -23638.098,E2 -23638.098} C_VEL
LIN {X 0,Y 157.318,Z 330.895,A -85,B 0,C 180,E1 -23643.458,E2 -23643.458} C_VEL
LIN {X 0,Y 157.367,Z 330.885,A -85,B 0,C 180,E1 -23649.695,E2 -23649.695} C_VEL
LIN {X 0,Y 157.495,Z 331.005,A -85,B 0,C 180,E1 -23655.579,E2 -23655.579} C_VEL
LIN {X 0,Y 158.431,Z 333.64,A -85,B 0,C 180,E1 -23656.007,E2 -23656.007} C_VEL
LIN {X 0,Y 160.227,Z 336.212,A -85,B 0,C 180,E1 -23656.659,E2 -23656.659} C_VEL
LIN {X 0,Y 164.88,Z 343.681,A -85,B 0,C 180,E1 -23658.306,E2 -23658.306} C_VEL
LIN {X 0,Y 171.647,Z 356.272,A -85,B 0,C 180,E1 -23660.612,E2 -23660.612} C_VEL
LIN {X 0,Y 176.856,Z 366.3,A -85,B 0,C 180,E1 -23662.262,E2 -23662.262} C_VEL
LIN {X 0,Y 180.773,Z 376.942,A -85,B 0,C 180,E1 -23663.58,E2 -23663.58} C_VEL
LIN {X 0,Y 178.11,Z 422.053,A -85,B 0,C 180,E1 -23665.378,E2 -23665.378} C_VEL
LIN {X 0,Y 177.015,Z 435.503,A -85,B 0,C 180,E1 -23666.096,E2 -23666.096} C_VEL
LIN {X 0,Y 175.364,Z 448.984,A -85,B 0,C 180,E1 -23667.282,E2 -23667.282} C_VEL
LIN {X 0,Y 173.221,Z 461.456,A -85,B 0,C 180,E1 -23668.83,E2 -23668.83} C_VEL
LIN {X 0,Y 170.537,Z 473.651,A -85,B 0,C 180,E1 -23670.878,E2 -23670.878} C_VEL
LIN {X 0,Y 167.684,Z 484.736,A -85,B 0,C 180,E1 -23673.296,E2 -23673.296} C_VEL
LIN {X 0,Y 164.85,Z 494.723,A -85,B 0,C 180,E1 -23676.11,E2 -23676.11} C_VEL
LIN {X 0,Y 162.042,Z 504.005,A -85,B 0,C 180,E1 -23679.442,E2 -23679.442} C_VEL
LIN {X 0,Y 159.546,Z 512.255,A -85,B 0,C 180,E1 -23683.235,E2 -23683.235} C_VEL
LIN {X 0,Y 157.369,Z 519.393,A -85,B 0,C 180,E1 -23687.535,E2 -23687.535} C_VEL
LIN {X 0,Y 156.18,Z 523.954,A -85,B 0,C 180,E1 -23691.089,E2 -23691.089} C_VEL
LIN {X 0,Y 155.175,Z 527.873,A -85,B 0,C 180,E1 -23695.066,E2 -23695.066} C_VEL
LIN {X 0,Y 154.436,Z 531.322,A -85,B 0,C 180,E1 -23700.157,E2 -23700.157} C_VEL
LIN {X 0,Y 154.587,Z 533.085,A -85,B 0,C 180,E1 -23705.081,E2 -23705.081} C_VEL
LIN {X 0,Y 155.456,Z 533.472,A -85,B 0,C 180,E1 -23709.776,E2 -23709.776} C_VEL
LIN {X 0,Y 157.016,Z 532.631,A -85,B 0,C 180,E1 -23714.262,E2 -23714.262} C_VEL
LIN {X 0,Y 159.216,Z 530.624,A -85,B 0,C 180,E1 -23718.608,E2 -23718.608} C_VEL
LIN {X 0,Y 162.78,Z 526.674,A -85,B 0,C 180,E1 -23723.515,E2 -23723.515} C_VEL
LIN {X 0,Y 166.648,Z 521.909,A -85,B 0,C 180,E1 -23727.486,E2 -23727.486} C_VEL
LIN {X 0,Y 170.808,Z 516.251,A -85,B 0,C 180,E1 -23730.945,E2 -23730.945} C_VEL
LIN {X 0,Y 175.981,Z 508.336,A -85,B 0,C 180,E1 -23734.533,E2 -23734.533} C_VEL
LIN {X 0,Y 180.819,Z 499.969,A -85,B 0,C 180,E1 -23737.423,E2 -23737.423} C_VEL
LIN {X 0,Y 185.707,Z 490.469,A -85,B 0,C 180,E1 -23739.935,E2 -23739.935} C_VEL
LIN {X 0,Y 190.255,Z 480.243,A -85,B 0,C 180,E1 -23741.992,E2 -23741.992} C_VEL
LIN {X 0,Y 194.372,Z 469.109,A -85,B 0,C 180,E1 -23743.739,E2 -23743.739} C_VEL
LIN {X 0,Y 197.63,Z 458.383,A -85,B 0,C 180,E1 -23745.022,E2 -23745.022} C_VEL
LIN {X 0,Y 200.552,Z 445.422,A -85,B 0,C 180,E1 -23746.201,E2 -23746.201} C_VEL
LIN {X 0,Y 202.554,Z 433.483,A -85,B 0,C 180,E1 -23746.908,E2 -23746.908} C_VEL
LIN {X 0,Y 204.875,Z 409.097,A -85,B 0,C 180,E1 -23747.797,E2 -23747.797} C_VEL
LIN {X 0,Y 206.039,Z 395.039,A -85,B 0,C 180,E1 -23748.295,E2 -23748.295} C_VEL
LIN {X 0,Y 202.959,Z 388.571,A -85,B 0,C 180,E1 -23750.14,E2 -23750.14} C_VEL
LIN {X 0,Y 198.896,Z 381.249,A -85,B 0,C 180,E1 -23752.757,E2 -23752.757} C_VEL
LIN {X 0,Y 194.426,Z 373.787,A -85,B 0,C 180,E1 -23756.146,E2 -23756.146} C_VEL
LIN {X 0,Y 191.841,Z 369.913,A -85,B 0,C 180,E1 -23758.437,E2 -23758.437} C_VEL
LIN {X 0,Y 189.265,Z 366.064,A -85,B 0,C 180,E1 -23761.103,E2 -23761.103} C_VEL
LIN {X 0,Y 188.516,Z 364.929,A -85,B 0,C 180,E1 -23762.008,E2 -23762.008} C_VEL
LIN {X 0,Y 186.393,Z 361.875,A -85,B 0,C 180,E1 -23764.968,E2 -23764.968} C_VEL
LIN {X 0,Y 186.076,Z 361.111,A -85,B 0,C 180,E1 -23765.543,E2 -23765.543} C_VEL
LIN {X 0,Y 183.14,Z 358.918,A -85,B 0,C 180,E1 -23772.744,E2 -23772.744} C_VEL
LIN {X 0,Y 182.867,Z 358.607,A -85,B 0,C 180,E1 -23776.134,E2 -23776.134} C_VEL
LIN {X 0,Y 183.578,Z 359.647,A -85,B 0,C 180,E1 -23780.801,E2 -23780.801} C_VEL
LIN {X 0,Y 185.222,Z 361.141,A -85,B 0,C 180,E1 -23784.669,E2 -23784.669} C_VEL
LIN {X 0,Y 186.316,Z 362.852,A -85,B 0,C 180,E1 -23786.585,E2 -23786.585} C_VEL
LIN {X 0,Y 189.703,Z 368.454,A -85,B 0,C 180,E1 -23791.082,E2 -23791.082} C_VEL
LIN {X 0,Y 192.888,Z 374.098,A -85,B 0,C 180,E1 -23794.314,E2 -23794.314} C_VEL
LIN {X 0,Y 195.42,Z 378.855,A -85,B 0,C 180,E1 -23796.463,E2 -23796.463} C_VEL
LIN {X 0,Y 198.949,Z 385.975,A -85,B 0,C 180,E1 -23799.141,E2 -23799.141} C_VEL
LIN {X 0,Y 203.023,Z 395.637,A -85,B 0,C 180,E1 -23801.9,E2 -23801.9} C_VEL
LIN {X 0,Y 205.533,Z 402.873,A -85,B 0,C 180,E1 -23803.511,E2 -23803.511} C_VEL
LIN {X 0,Y 202.157,Z 440.159,A -85,B 0,C 180,E1 -23804.807,E2 -23804.807} C_VEL
LIN {X 0,Y 199.827,Z 453.968,A -85,B 0,C 180,E1 -23805.577,E2 -23805.577} C_VEL
LIN {X 0,Y 196.733,Z 466.379,A -85,B 0,C 180,E1 -23806.566,E2 -23806.566} C_VEL
LIN {X 0,Y 192.8,Z 478.647,A -85,B 0,C 180,E1 -23807.96,E2 -23807.96} C_VEL
LIN {X 0,Y 188.504,Z 489.698,A -85,B 0,C 180,E1 -23809.637,E2 -23809.637} C_VEL
LIN {X 0,Y 183.94,Z 499.763,A -85,B 0,C 180,E1 -23811.632,E2 -23811.632} C_VEL
LIN {X 0,Y 179.16,Z 508.892,A -85,B 0,C 180,E1 -23813.967,E2 -23813.967} C_VEL
LIN {X 0,Y 174.025,Z 517.846,A -85,B 0,C 180,E1 -23816.974,E2 -23816.974} C_VEL
LIN {X 0,Y 171.966,Z 521.101,A -85,B 0,C 180,E1 -23818.287,E2 -23818.287} C_VEL
LIN {X 0,Y 169.223,Z 524.432,A -85,B 0,C 180,E1 -23819.658,E2 -23819.658} C_VEL
LIN {X 0,Y 163.32,Z 529.439,A -85,B 0,C 180,E1 -23821.816,E2 -23821.816} C_VEL
LIN {X 0,Y 157.637,Z 533.73,A -85,B 0,C 180,E1 -23824.274,E2 -23824.274} C_VEL
LIN {X 0,Y 155.309,Z 535.911,A -85,B 0,C 180,E1 -23826.091,E2 -23826.091} C_VEL
LIN {X 0,Y 151.579,Z 540.25,A -85,B 0,C 180,E1 -23831.072,E2 -23831.072} C_VEL
LIN {X 0,Y 150.149,Z 541.862,A -85,B 0,C 180,E1 -23833.7,E2 -23833.7} C_VEL
LIN {X 0,Y 149.119,Z 543.057,A -85,B 0,C 180,E1 -23836.38,E2 -23836.38} C_VEL
LIN {X 0,Y 147.902,Z 544.258,A -85,B 0,C 180,E1 -23841.814,E2 -23841.814} C_VEL
LIN {X 0,Y 147.686,Z 544.293,A -85,B 0,C 180,E1 -23844.548,E2 -23844.548} C_VEL
LIN {X 0,Y 147.694,Z 543.8,A -85,B 0,C 180,E1 -23847.829,E2 -23847.829} C_VEL
LIN {X 0,Y 147.87,Z 543.152,A -85,B 0,C 180,E1 -23850.009,E2 -23850.009} C_VEL
LIN {X 0,Y 147.757,Z 541.927,A -85,B 0,C 180,E1 -23852.735,E2 -23852.735} C_VEL
LIN {X 0,Y 147.848,Z 539.269,A -85,B 0,C 180,E1 -23856.834,E2 -23856.834} C_VEL
LIN {X 0,Y 148.383,Z 535.545,A -85,B 0,C 180,E1 -23860.929,E2 -23860.929} C_VEL
LIN {X 0,Y 149.459,Z 530.652,A -85,B 0,C 180,E1 -23864.997,E2 -23864.997} C_VEL
LIN {X 0,Y 151.283,Z 524.461,A -85,B 0,C 180,E1 -23868.985,E2 -23868.985} C_VEL
LIN {X 0,Y 153.775,Z 516.732,A -85,B 0,C 180,E1 -23872.867,E2 -23872.867} C_VEL
LIN {X 0,Y 155.379,Z 511.266,A -85,B 0,C 180,E1 -23875.103,E2 -23875.103} C_VEL
LIN {X 0,Y 157.88,Z 503.152,A -85,B 0,C 180,E1 -23877.873,E2 -23877.873} C_VEL
LIN {X 0,Y 160.868,Z 493.358,A -85,B 0,C 180,E1 -23880.529,E2 -23880.529} C_VEL
LIN {X 0,Y 163.771,Z 482.629,A -85,B 0,C 180,E1 -23882.812,E2 -23882.812} C_VEL
LIN {X 0,Y 166.516,Z 470.642,A -85,B 0,C 180,E1 -23884.742,E2 -23884.742} C_VEL
LIN {X 0,Y 168.861,Z 458.308,A -85,B 0,C 180,E1 -23886.198,E2 -23886.198} C_VEL
LIN {X 0,Y 170.596,Z 445.714,A -85,B 0,C 180,E1 -23887.241,E2 -23887.241} C_VEL
LIN {X 0,Y 171.792,Z 430.02,A -85,B 0,C 180,E1 -23888.029,E2 -23888.029} C_VEL
LIN {X 0,Y 173.783,Z 396.749,A -85,B 0,C 180,E1 -23889.405,E2 -23889.405} C_VEL
LIN {X 0,Y 172.474,Z 382.402,A -85,B 0,C 180,E1 -23890.44,E2 -23890.44} C_VEL
LIN {X 0,Y 165.775,Z 364.313,A -85,B 0,C 180,E1 -23892.947,E2 -23892.947} C_VEL
LIN {X 0,Y 159.297,Z 349.627,A -85,B 0,C 180,E1 -23895.423,E2 -23895.423} C_VEL
LIN {X 0,Y 153.764,Z 338.873,A -85,B 0,C 180,E1 -23897.651,E2 -23897.651} C_VEL
LIN {X 0,Y 152.194,Z 335.967,A -85,B 0,C 180,E1 -23898.316,E2 -23898.316} C_VEL
LIN {X 0,Y 150.521,Z 333.279,A -85,B 0,C 180,E1 -23899.015,E2 -23899.015} C_VEL
LIN {X 0,Y 150.162,Z 331.779,A -85,B 0,C 180,E1 -23899.284,E2 -23899.284} C_VEL
LIN {X 0,Y 150.186,Z 331.778,A -85,B 0,C 180,E1 -23902.713,E2 -23902.713} C_VEL
LIN {X 0,Y 150.225,Z 331.776,A -85,B 0,C 180,E1 -23907.372,E2 -23907.372} C_VEL
LIN {X 0,Y 150.253,Z 331.77,A -85,B 0,C 180,E1 -23912.723,E2 -23912.723} C_VEL
LIN {X 0,Y 150.296,Z 331.758,A -85,B 0,C 180,E1 -23919.278,E2 -23919.278} C_VEL
LIN {X 0,Y 150.327,Z 331.717,A -85,B 0,C 180,E1 -23923.709,E2 -23923.709} C_VEL
LIN {X 0,Y 150.618,Z 331.721,A -85,B 0,C 180,E1 -23929.243,E2 -23929.243} C_VEL
LIN {X 0,Y 150.694,Z 331.709,A -85,B 0,C 180,E1 -23931.957,E2 -23931.957} C_VEL
LIN {X 0,Y 151.216,Z 331.604,A -85,B 0,C 180,E1 -23940,E2 -23940} C_VEL
LIN {X 0,Y 150.688,Z 331.709,A -85,B 0,C 180,E1 -23948.043,E2 -23948.043} C_VEL
LIN {X 0,Y 150.583,Z 331.715,A -85,B 0,C 180,E1 -23951.422,E2 -23951.422} C_VEL
LIN {X 0,Y 150.326,Z 331.755,A -85,B 0,C 180,E1 -23956.291,E2 -23956.291} C_VEL
LIN {X 0,Y 150.293,Z 331.754,A -85,B 0,C 180,E1 -23960.719,E2 -23960.719} C_VEL
LIN {X 0,Y 150.19,Z 331.754,A -85,B 0,C 180,E1 -23967.23,E2 -23967.23} C_VEL
LIN {X 0,Y 150.194,Z 331.721,A -85,B 0,C 180,E1 -23972.609,E2 -23972.609} C_VEL
LIN {X 0,Y 150.179,Z 331.774,A -85,B 0,C 180,E1 -23977.472,E2 -23977.472} C_VEL
LIN {X 0,Y 150.142,Z 331.776,A -85,B 0,C 180,E1 -23981.492,E2 -23981.492} C_VEL
LIN {X 0,Y 150.137,Z 331.783,A -85,B 0,C 180,E1 -23985.391,E2 -23985.391} C_VEL
LIN {X 0,Y 150.145,Z 331.772,A -85,B 0,C 180,E1 -23989.049,E2 -23989.049} C_VEL
LIN {X 0,Y 150.185,Z 331.78,A -85,B 0,C 180,E1 -23992.705,E2 -23992.705} C_VEL
LIN {X 0,Y 150.217,Z 331.775,A -85,B 0,C 180,E1 -23997.368,E2 -23997.368} C_VEL
LIN {X 0,Y 150.247,Z 331.772,A -85,B 0,C 180,E1 -24002.717,E2 -24002.717} C_VEL
LIN {X 0,Y 150.292,Z 331.768,A -85,B 0,C 180,E1 -24009.269,E2 -24009.269} C_VEL
LIN {X 0,Y 150.334,Z 331.761,A -85,B 0,C 180,E1 -24013.441,E2 -24013.441} C_VEL
LIN {X 0,Y 151.408,Z 334.699,A -85,B 0,C 180,E1 -24014.029,E2 -24014.029} C_VEL
LIN {X 0,Y 153.04,Z 336.781,A -85,B 0,C 180,E1 -24014.662,E2 -24014.662} C_VEL
LIN {X 0,Y 161.21,Z 350.049,A -85,B 0,C 180,E1 -24017.767,E2 -24017.767} C_VEL
LIN {X 0,Y 171.167,Z 369.257,A -85,B 0,C 180,E1 -24021.221,E2 -24021.221} C_VEL
LIN {X 0,Y 174.693,Z 378.836,A -85,B 0,C 180,E1 -24022.484,E2 -24022.484} C_VEL
LIN {X 0,Y 171.324,Z 430.639,A -85,B 0,C 180,E1 -24024.662,E2 -24024.662} C_VEL
LIN {X 0,Y 169.779,Z 444.372,A -85,B 0,C 180,E1 -24025.708,E2 -24025.708} C_VEL
LIN {X 0,Y 167.726,Z 457.063,A -85,B 0,C 180,E1 -24027.144,E2 -24027.144} C_VEL
LIN {X 0,Y 165.113,Z 469.504,A -85,B 0,C 180,E1 -24029.078,E2 -24029.078} C_VEL
LIN {X 0,Y 162.295,Z 480.628,A -85,B 0,C 180,E1 -24031.34,E2 -24031.34} C_VEL
LIN {X 0,Y 159.29,Z 491.088,A -85,B 0,C 180,E1 -24034.103,E2 -24034.103} C_VEL
LIN {X 0,Y 156.593,Z 499.937,A -85,B 0,C 180,E1 -24037.068,E2 -24037.068} C_VEL
LIN {X 0,Y 153.953,Z 508.135,A -85,B 0,C 180,E1 -24040.512,E2 -24040.512} C_VEL
LIN {X 0,Y 151.972,Z 514.372,A -85,B 0,C 180,E1 -24043.794,E2 -24043.794} C_VEL
LIN {X 0,Y 150.147,Z 520.315,A -85,B 0,C 180,E1 -24047.703,E2 -24047.703} C_VEL
LIN {X 0,Y 148.743,Z 525.541,A -85,B 0,C 180,E1 -24052.198,E2 -24052.198} C_VEL
LIN {X 0,Y 147.717,Z 529.455,A -85,B 0,C 180,E1 -24056.864,E2 -24056.864} C_VEL
LIN {X 0,Y 147.284,Z 532.114,A -85,B 0,C 180,E1 -24061.648,E2 -24061.648} C_VEL
LIN {X 0,Y 147.575,Z 533.424,A -85,B 0,C 180,E1 -24065.943,E2 -24065.943} C_VEL
LIN {X 0,Y 148.79,Z 533.71,A -85,B 0,C 180,E1 -24071.382,E2 -24071.382} C_VEL
LIN {X 0,Y 150.403,Z 532.84,A -85,B 0,C 180,E1 -24075.499,E2 -24075.499} C_VEL
LIN {X 0,Y 152.786,Z 530.823,A -85,B 0,C 180,E1 -24079.91,E2 -24079.91} C_VEL
LIN {X 0,Y 155.987,Z 527.604,A -85,B 0,C 180,E1 -24084.173,E2 -24084.173} C_VEL
LIN {X 0,Y 159.849,Z 523.221,A -85,B 0,C 180,E1 -24088.156,E2 -24088.156} C_VEL
LIN {X 0,Y 164.474,Z 517.438,A -85,B 0,C 180,E1 -24091.964,E2 -24091.964} C_VEL
LIN {X 0,Y 169.778,Z 510.036,A -85,B 0,C 180,E1 -24095.574,E2 -24095.574} C_VEL
LIN {X 0,Y 174.98,Z 501.684,A -85,B 0,C 180,E1 -24098.62,E2 -24098.62} C_VEL
LIN {X 0,Y 179.791,Z 492.915,A -85,B 0,C 180,E1 -24101.089,E2 -24101.089} C_VEL
LIN {X 0,Y 184.477,Z 483.366,A -85,B 0,C 180,E1 -24103.135,E2 -24103.135} C_VEL
LIN {X 0,Y 188.623,Z 473.173,A -85,B 0,C 180,E1 -24104.881,E2 -24104.881} C_VEL
LIN {X 0,Y 192.498,Z 461.623,A -85,B 0,C 180,E1 -24106.38,E2 -24106.38} C_VEL
LIN {X 0,Y 195.631,Z 449.65,A -85,B 0,C 180,E1 -24107.552,E2 -24107.552} C_VEL
LIN {X 0,Y 197.968,Z 437.509,A -85,B 0,C 180,E1 -24108.401,E2 -24108.401} C_VEL
LIN {X 0,Y 199.742,Z 423.323,A -85,B 0,C 180,E1 -24108.988,E2 -24108.988} C_VEL
LIN {X 0,Y 201.982,Z 398.142,A -85,B 0,C 180,E1 -24109.865,E2 -24109.865} C_VEL
LIN {X 0,Y 197.827,Z 389.738,A -85,B 0,C 180,E1 -24112.604,E2 -24112.604} C_VEL
LIN {X 0,Y 193.706,Z 382.496,A -85,B 0,C 180,E1 -24115.737,E2 -24115.737} C_VEL
LIN {X 0,Y 191.493,Z 378.857,A -85,B 0,C 180,E1 -24117.663,E2 -24117.663} C_VEL
LIN {X 0,Y 189.885,Z 376.273,A -85,B 0,C 180,E1 -24119.238,E2 -24119.238} C_VEL
LIN {X 0,Y 187.39,Z 372.112,A -85,B 0,C 180,E1 -24122.085,E2 -24122.085} C_VEL
LIN {X 0,Y 184.957,Z 368.518,A -85,B 0,C 180,E1 -24125.607,E2 -24125.607} C_VEL
LIN {X 0,Y 184.713,Z 367.963,A -85,B 0,C 180,E1 -24126.069,E2 -24126.069} C_VEL
LIN {X 0,Y 182.136,Z 365.937,A -85,B 0,C 180,E1 -24132.816,E2 -24132.816} C_VEL
LIN {X 0,Y 181.908,Z 365.709,A -85,B 0,C 180,E1 -24136.762,E2 -24136.762} C_VEL
LIN {X 0,Y 183.785,Z 367.69,A -85,B 0,C 180,E1 -24143.784,E2 -24143.784} C_VEL
LIN {X 0,Y 184.986,Z 369.685,A -85,B 0,C 180,E1 -24146.128,E2 -24146.128} C_VEL
LIN {X 0,Y 188.018,Z 375.082,A -85,B 0,C 180,E1 -24150.444,E2 -24150.444} C_VEL
LIN {X 0,Y 190.879,Z 380.395,A -85,B 0,C 180,E1 -24153.524,E2 -24153.524} C_VEL
LIN {X 0,Y 193.323,Z 385.372,A -85,B 0,C 180,E1 -24155.771,E2 -24155.771} C_VEL
LIN {X 0,Y 196.335,Z 391.861,A -85,B 0,C 180,E1 -24158.226,E2 -24158.226} C_VEL
LIN {X 0,Y 199.877,Z 400.779,A -85,B 0,C 180,E1 -24160.811,E2 -24160.811} C_VEL
LIN {X 0,Y 201.425,Z 405.448,A -85,B 0,C 180,E1 -24161.906,E2 -24161.906} C_VEL
LIN {X 0,Y 198.126,Z 440.183,A -85,B 0,C 180,E1 -24163.14,E2 -24163.14} C_VEL
LIN {X 0,Y 195.601,Z 454.307,A -85,B 0,C 180,E1 -24163.931,E2 -24163.931} C_VEL
LIN {X 0,Y 192.314,Z 466.769,A -85,B 0,C 180,E1 -24164.937,E2 -24164.937} C_VEL
LIN {X 0,Y 188.231,Z 478.908,A -85,B 0,C 180,E1 -24166.325,E2 -24166.325} C_VEL
LIN {X 0,Y 183.769,Z 489.866,A -85,B 0,C 180,E1 -24168.003,E2 -24168.003} C_VEL
LIN {X 0,Y 178.484,Z 500.804,A -85,B 0,C 180,E1 -24170.231,E2 -24170.231} C_VEL
LIN {X 0,Y 173.514,Z 509.709,A -85,B 0,C 180,E1 -24172.599,E2 -24172.599} C_VEL
LIN {X 0,Y 168.158,Z 518.448,A -85,B 0,C 180,E1 -24175.664,E2 -24175.664} C_VEL
LIN {X 0,Y 163.236,Z 525.531,A -85,B 0,C 180,E1 -24178.904,E2 -24178.904} C_VEL
LIN {X 0,Y 158.679,Z 531.768,A -85,B 0,C 180,E1 -24182.755,E2 -24182.755} C_VEL
LIN {X 0,Y 155.309,Z 535.911,A -85,B 0,C 180,E1 -24186.091,E2 -24186.091} C_VEL
LIN {X 0,Y 153.101,Z 537.885,A -85,B 0,C 180,E1 -24187.999,E2 -24187.999} C_VEL
LIN {X 0,Y 148.034,Z 540.562,A -85,B 0,C 180,E1 -24191.082,E2 -24191.082} C_VEL
LIN {X 0,Y 143.374,Z 542.445,A -85,B 0,C 180,E1 -24194.437,E2 -24194.437} C_VEL
LIN {X 0,Y 141.872,Z 543.175,A -85,B 0,C 180,E1 -24196.706,E2 -24196.706} C_VEL
LIN {X 0,Y 140.851,Z 544.014,A -85,B 0,C 180,E1 -24201.401,E2 -24201.401} C_VEL
LIN {X 0,Y 140.615,Z 543.999,A -85,B 0,C 180,E1 -24204.273,E2 -24204.273} C_VEL
LIN {X 0,Y 140.634,Z 543.307,A -85,B 0,C 180,E1 -24208.145,E2 -24208.145} C_VEL
LIN {X 0,Y 140.775,Z 542.722,A -85,B 0,C 180,E1 -24210.009,E2 -24210.009} C_VEL
LIN {X 0,Y 140.658,Z 541.452,A -85,B 0,C 180,E1 -24212.873,E2 -24212.873} C_VEL
LIN {X 0,Y 140.783,Z 538.697,A -85,B 0,C 180,E1 -24217.178,E2 -24217.178} C_VEL
LIN {X 0,Y 141.383,Z 534.867,A -85,B 0,C 180,E1 -24221.477,E2 -24221.477} C_VEL
LIN {X 0,Y 142.574,Z 529.862,A -85,B 0,C 180,E1 -24225.739,E2 -24225.739} C_VEL
LIN {X 0,Y 144.548,Z 523.547,A -85,B 0,C 180,E1 -24229.906,E2 -24229.906} C_VEL
LIN {X 0,Y 147.183,Z 515.603,A -85,B 0,C 180,E1 -24233.954,E2 -24233.954} C_VEL
LIN {X 0,Y 148.601,Z 511.004,A -85,B 0,C 180,E1 -24235.898,E2 -24235.898} C_VEL
LIN {X 0,Y 151.571,Z 501.749,A -85,B 0,C 180,E1 -24239.142,E2 -24239.142} C_VEL
LIN {X 0,Y 154.679,Z 491.692,A -85,B 0,C 180,E1 -24241.891,E2 -24241.891} C_VEL
LIN {X 0,Y 157.872,Z 480.574,A -85,B 0,C 180,E1 -24244.203,E2 -24244.203} C_VEL
LIN {X 0,Y 160.273,Z 470.079,A -85,B 0,C 180,E1 -24245.916,E2 -24245.916} C_VEL
LIN {X 0,Y 162.706,Z 457.658,A -85,B 0,C 180,E1 -24247.41,E2 -24247.41} C_VEL
LIN {X 0,Y 164.499,Z 444.798,A -85,B 0,C 180,E1 -24248.481,E2 -24248.481} C_VEL
LIN {X 0,Y 165.771,Z 428.496,A -85,B 0,C 180,E1 -24249.3,E2 -24249.3} C_VEL
LIN {X 0,Y 167.719,Z 396.226,A -85,B 0,C 180,E1 -24250.687,E2 -24250.687} C_VEL
LIN {X 0,Y 166.543,Z 384.568,A -85,B 0,C 180,E1 -24251.604,E2 -24251.604} C_VEL
LIN {X 0,Y 160.393,Z 367.734,A -85,B 0,C 180,E1 -24254.038,E2 -24254.038} C_VEL
LIN {X 0,Y 154.421,Z 353.88,A -85,B 0,C 180,E1 -24256.485,E2 -24256.485} C_VEL
LIN {X 0,Y 148.029,Z 341.206,A -85,B 0,C 180,E1 -24259.246,E2 -24259.246} C_VEL
LIN {X 0,Y 145.826,Z 337.724,A -85,B 0,C 180,E1 -24260.202,E2 -24260.202} C_VEL
LIN {X 0,Y 143.673,Z 334.646,A -85,B 0,C 180,E1 -24261.151,E2 -24261.151} C_VEL
LIN {X 0,Y 143.11,Z 332.66,A -85,B 0,C 180,E1 -24261.569,E2 -24261.569} C_VEL
LIN {X 0,Y 143.192,Z 332.653,A -85,B 0,C 180,E1 -24267.324,E2 -24267.324} C_VEL
LIN {X 0,Y 143.2,Z 332.65,A -85,B 0,C 180,E1 -24272.068,E2 -24272.068} C_VEL
LIN {X 0,Y 143.237,Z 332.639,A -85,B 0,C 180,E1 -24278.802,E2 -24278.802} C_VEL
LIN {X 0,Y 143.266,Z 332.597,A -85,B 0,C 180,E1 -24282.882,E2 -24282.882} C_VEL
LIN {X 0,Y 143.545,Z 332.6,A -85,B 0,C 180,E1 -24288.706,E2 -24288.706} C_VEL
LIN {X 0,Y 143.62,Z 332.591,A -85,B 0,C 180,E1 -24291.558,E2 -24291.558} C_VEL
LIN {X 0,Y 144.174,Z 332.479,A -85,B 0,C 180,E1 -24300,E2 -24300} C_VEL
LIN {X 0,Y 143.614,Z 332.589,A -85,B 0,C 180,E1 -24308.442,E2 -24308.442} C_VEL
LIN {X 0,Y 143.508,Z 332.596,A -85,B 0,C 180,E1 -24311.608,E2 -24311.608} C_VEL
LIN {X 0,Y 143.266,Z 332.63,A -85,B 0,C 180,E1 -24317.118,E2 -24317.118} C_VEL
LIN {X 0,Y 143.23,Z 332.637,A -85,B 0,C 180,E1 -24321.19,E2 -24321.19} C_VEL
LIN {X 0,Y 143.12,Z 332.627,A -85,B 0,C 180,E1 -24327.871,E2 -24327.871} C_VEL
LIN {X 0,Y 143.13,Z 332.606,A -85,B 0,C 180,E1 -24333.401,E2 -24333.401} C_VEL
LIN {X 0,Y 143.082,Z 332.66,A -85,B 0,C 180,E1 -24338.186,E2 -24338.186} C_VEL
LIN {X 0,Y 143.044,Z 332.656,A -85,B 0,C 180,E1 -24343.46,E2 -24343.46} C_VEL
LIN {X 0,Y 143.047,Z 332.664,A -85,B 0,C 180,E1 -24347.474,E2 -24347.474} C_VEL
LIN {X 0,Y 143.081,Z 332.663,A -85,B 0,C 180,E1 -24351.805,E2 -24351.805} C_VEL
LIN {X 0,Y 143.184,Z 332.65,A -85,B 0,C 180,E1 -24357.314,E2 -24357.314} C_VEL
LIN {X 0,Y 143.191,Z 332.648,A -85,B 0,C 180,E1 -24362.063,E2 -24362.063} C_VEL
LIN {X 0,Y 143.233,Z 332.651,A -85,B 0,C 180,E1 -24368.792,E2 -24368.792} C_VEL
LIN {X 0,Y 143.275,Z 332.638,A -85,B 0,C 180,E1 -24371.212,E2 -24371.212} C_VEL
LIN {X 0,Y 144.22,Z 335.351,A -85,B 0,C 180,E1 -24371.75,E2 -24371.75} C_VEL
LIN {X 0,Y 146.151,Z 337.981,A -85,B 0,C 180,E1 -24372.592,E2 -24372.592} C_VEL
LIN {X 0,Y 155.044,Z 352.076,A -85,B 0,C 180,E1 -24376.238,E2 -24376.238} C_VEL
LIN {X 0,Y 165.678,Z 372.574,A -85,B 0,C 180,E1 -24380.173,E2 -24380.173} C_VEL
LIN {X 0,Y 167.711,Z 378.091,A -85,B 0,C 180,E1 -24380.95,E2 -24380.95} C_VEL
LIN {X 0,Y 168.542,Z 380.365,A -85,B 0,C 180,E1 -24381.263,E2 -24381.263} C_VEL
LIN {X 0,Y 165.198,Z 430.667,A -85,B 0,C 180,E1 -24383.443,E2 -24383.443} C_VEL
LIN {X 0,Y 163.589,Z 444.508,A -85,B 0,C 180,E1 -24384.522,E2 -24384.522} C_VEL
LIN {X 0,Y 161.705,Z 456.045,A -85,B 0,C 180,E1 -24385.839,E2 -24385.839} C_VEL
LIN {X 0,Y 159.032,Z 468.503,A -85,B 0,C 180,E1 -24387.776,E2 -24387.776} C_VEL
LIN {X 0,Y 156.158,Z 479.4,A -85,B 0,C 180,E1 -24389.992,E2 -24389.992} C_VEL
LIN {X 0,Y 152.894,Z 490.57,A -85,B 0,C 180,E1 -24392.955,E2 -24392.955} C_VEL
LIN {X 0,Y 150.097,Z 499.417,A -85,B 0,C 180,E1 -24395.977,E2 -24395.977} C_VEL
LIN {X 0,Y 147.232,Z 507.86,A -85,B 0,C 180,E1 -24399.608,E2 -24399.608} C_VEL
LIN {X 0,Y 144.743,Z 515.472,A -85,B 0,C 180,E1 -24403.806,E2 -24403.806} C_VEL
LIN {X 0,Y 142.657,Z 522.05,A -85,B 0,C 180,E1 -24408.605,E2 -24408.605} C_VEL
LIN {X 0,Y 141.298,Z 526.99,A -85,B 0,C 180,E1 -24413.436,E2 -24413.436} C_VEL
LIN {X 0,Y 140.647,Z 529.52,A -85,B 0,C 180,E1 -24416.713,E2 -24416.713} C_VEL
LIN {X 0,Y 140.189,Z 532.169,A -85,B 0,C 180,E1 -24421.542,E2 -24421.542} C_VEL
LIN {X 0,Y 140.596,Z 533.757,A -85,B 0,C 180,E1 -24426.889,E2 -24426.889} C_VEL
LIN {X 0,Y 141.851,Z 534.007,A -85,B 0,C 180,E1 -24431.997,E2 -24431.997} C_VEL
LIN {X 0,Y 143.955,Z 532.961,A -85,B 0,C 180,E1 -24437.063,E2 -24437.063} C_VEL
LIN {X 0,Y 146.494,Z 530.959,A -85,B 0,C 180,E1 -24441.415,E2 -24441.415} C_VEL
LIN {X 0,Y 149.991,Z 527.721,A -85,B 0,C 180,E1 -24445.787,E2 -24445.787} C_VEL
LIN {X 0,Y 154.257,Z 523.233,A -85,B 0,C 180,E1 -24449.933,E2 -24449.933} C_VEL
LIN {X 0,Y 159.213,Z 517.407,A -85,B 0,C 180,E1 -24453.805,E2 -24453.805} C_VEL
LIN {X 0,Y 164.818,Z 509.97,A -85,B 0,C 180,E1 -24457.432,E2 -24457.432} C_VEL
LIN {X 0,Y 169.76,Z 502.477,A -85,B 0,C 180,E1 -24460.203,E2 -24460.203} C_VEL
LIN {X 0,Y 174.795,Z 493.836,A -85,B 0,C 180,E1 -24462.692,E2 -24462.692} C_VEL
LIN {X 0,Y 180.384,Z 483.003,A -85,B 0,C 180,E1 -24465.029,E2 -24465.029} C_VEL
LIN {X 0,Y 184.892,Z 472.263,A -85,B 0,C 180,E1 -24466.817,E2 -24466.817} C_VEL
LIN {X 0,Y 188.84,Z 460.788,A -85,B 0,C 180,E1 -24468.258,E2 -24468.258} C_VEL
LIN {X 0,Y 192.162,Z 448.13,A -85,B 0,C 180,E1 -24469.463,E2 -24469.463} C_VEL
LIN {X 0,Y 194.472,Z 436.049,A -85,B 0,C 180,E1 -24470.236,E2 -24470.236} C_VEL
LIN {X 0,Y 196.436,Z 419.142,A -85,B 0,C 180,E1 -24470.88,E2 -24470.88} C_VEL
LIN {X 0,Y 198.019,Z 401.346,A -85,B 0,C 180,E1 -24471.533,E2 -24471.533} C_VEL
LIN {X 0,Y 194.096,Z 393.316,A -85,B 0,C 180,E1 -24474.434,E2 -24474.434} C_VEL
LIN {X 0,Y 190.108,Z 386.08,A -85,B 0,C 180,E1 -24477.881,E2 -24477.881} C_VEL
LIN {X 0,Y 188.024,Z 382.677,A -85,B 0,C 180,E1 -24480,E2 -24480} C_VEL
LIN {X 0,Y 185.452,Z 378.271,A -85,B 0,C 180,E1 -24483.216,E2 -24483.216} C_VEL
LIN {X 0,Y 183.396,Z 374.83,A -85,B 0,C 180,E1 -24486.602,E2 -24486.602} C_VEL
LIN {X 0,Y 181.049,Z 372.841,A -85,B 0,C 180,E1 -24493.468,E2 -24493.468} C_VEL
LIN {X 0,Y 180.924,Z 372.757,A -85,B 0,C 180,E1 -24496.856,E2 -24496.856} C_VEL
LIN {X 0,Y 182.764,Z 374.798,A -85,B 0,C 180,E1 -24503.764,E2 -24503.764} C_VEL
LIN {X 0,Y 183.717,Z 376.652,A -85,B 0,C 180,E1 -24505.764,E2 -24505.764} C_VEL
LIN {X 0,Y 186.377,Z 381.707,A -85,B 0,C 180,E1 -24509.815,E2 -24509.815} C_VEL
LIN {X 0,Y 188.812,Z 386.481,A -85,B 0,C 180,E1 -24512.613,E2 -24512.613} C_VEL
LIN {X 0,Y 191.16,Z 391.674,A -85,B 0,C 180,E1 -24514.98,E2 -24514.98} C_VEL
LIN {X 0,Y 193.59,Z 397.148,A -85,B 0,C 180,E1 -24517.092,E2 -24517.092} C_VEL
LIN {X 0,Y 196.765,Z 405.773,A -85,B 0,C 180,E1 -24519.659,E2 -24519.659} C_VEL
LIN {X 0,Y 197.513,Z 408.13,A -85,B 0,C 180,E1 -24520.233,E2 -24520.233} C_VEL
LIN {X 0,Y 194.452,Z 439.43,A -85,B 0,C 180,E1 -24521.351,E2 -24521.351} C_VEL
LIN {X 0,Y 191.857,Z 453.606,A -85,B 0,C 180,E1 -24522.125,E2 -24522.125} C_VEL
LIN {X 0,Y 188.705,Z 465.427,A -85,B 0,C 180,E1 -24523.053,E2 -24523.053} C_VEL
LIN {X 0,Y 184.43,Z 477.756,A -85,B 0,C 180,E1 -24524.412,E2 -24524.412} C_VEL
LIN {X 0,Y 179.752,Z 488.831,A -85,B 0,C 180,E1 -24526.067,E2 -24526.067} C_VEL
LIN {X 0,Y 174.756,Z 498.918,A -85,B 0,C 180,E1 -24528.055,E2 -24528.055} C_VEL
LIN {X 0,Y 169.99,Z 507.272,A -85,B 0,C 180,E1 -24530.16,E2 -24530.16} C_VEL
LIN {X 0,Y 164.206,Z 516.394,A -85,B 0,C 180,E1 -24533.201,E2 -24533.201} C_VEL
LIN {X 0,Y 158.849,Z 523.799,A -85,B 0,C 180,E1 -24536.437,E2 -24536.437} C_VEL
LIN {X 0,Y 153.949,Z 530.132,A -85,B 0,C 180,E1 -24540.156,E2 -24540.156} C_VEL
LIN {X 0,Y 150.155,Z 534.576,A -85,B 0,C 180,E1 -24543.611,E2 -24543.611} C_VEL
LIN {X 0,Y 146.793,Z 538.3,A -85,B 0,C 180,E1 -24547.491,E2 -24547.491} C_VEL
LIN {X 0,Y 144.879,Z 540.26,A -85,B 0,C 180,E1 -24550.161,E2 -24550.161} C_VEL
LIN {X 0,Y 143.313,Z 541.799,A -85,B 0,C 180,E1 -24552.899,E2 -24552.899} C_VEL
LIN {X 0,Y 141.872,Z 543.175,A -85,B 0,C 180,E1 -24556.706,E2 -24556.706} C_VEL
LIN {X 0,Y 140.598,Z 543.743,A -85,B 0,C 180,E1 -24559.039,E2 -24559.039} C_VEL
LIN {X 0,Y 137.146,Z 543.888,A -85,B 0,C 180,E1 -24562.876,E2 -24562.876} C_VEL
LIN {X 0,Y 134.59,Z 543.446,A -85,B 0,C 180,E1 -24566.063,E2 -24566.063} C_VEL
LIN {X 0,Y 133.644,Z 542.786,A -85,B 0,C 180,E1 -24568.558,E2 -24568.558} C_VEL
LIN {X 0,Y 133.628,Z 542.491,A -85,B 0,C 180,E1 -24569.4,E2 -24569.4} C_VEL
LIN {X 0,Y 133.571,Z 540.956,A -85,B 0,C 180,E1 -24573.026,E2 -24573.026} C_VEL
LIN {X 0,Y 133.742,Z 538.098,A -85,B 0,C 180,E1 -24577.558,E2 -24577.558} C_VEL
LIN {X 0,Y 134.409,Z 534.158,A -85,B 0,C 180,E1 -24582.082,E2 -24582.082} C_VEL
LIN {X 0,Y 136.015,Z 528.035,A -85,B 0,C 180,E1 -24587.293,E2 -24587.293} C_VEL
LIN {X 0,Y 138.257,Z 521.302,A -85,B 0,C 180,E1 -24591.634,E2 -24591.634} C_VEL
LIN {X 0,Y 140.602,Z 514.414,A -85,B 0,C 180,E1 -24595.151,E2 -24595.151} C_VEL
LIN {X 0,Y 143.508,Z 506.116,A -85,B 0,C 180,E1 -24598.529,E2 -24598.529} C_VEL
LIN {X 0,Y 146.472,Z 497.053,A -85,B 0,C 180,E1 -24601.461,E2 -24601.461} C_VEL
LIN {X 0,Y 149.497,Z 487.3,A -85,B 0,C 180,E1 -24603.943,E2 -24603.943} C_VEL
LIN {X 0,Y 152.373,Z 476.774,A -85,B 0,C 180,E1 -24606.028,E2 -24606.028} C_VEL
LIN {X 0,Y 155.232,Z 464.201,A -85,B 0,C 180,E1 -24607.889,E2 -24607.889} C_VEL
LIN {X 0,Y 157.494,Z 451.308,A -85,B 0,C 180,E1 -24609.254,E2 -24609.254} C_VEL
LIN {X 0,Y 159.087,Z 438.031,A -85,B 0,C 180,E1 -24610.147,E2 -24610.147} C_VEL
LIN {X 0,Y 161.731,Z 397.242,A -85,B 0,C 180,E1 -24611.969,E2 -24611.969} C_VEL
LIN {X 0,Y 160.74,Z 386.997,A -85,B 0,C 180,E1 -24612.801,E2 -24612.801} C_VEL
LIN {X 0,Y 155.141,Z 371.31,A -85,B 0,C 180,E1 -24615.171,E2 -24615.171} C_VEL
LIN {X 0,Y 149.132,Z 357.212,A -85,B 0,C 180,E1 -24617.813,E2 -24617.813} C_VEL
LIN {X 0,Y 143.413,Z 345.826,A -85,B 0,C 180,E1 -24620.426,E2 -24620.426} C_VEL
LIN {X 0,Y 139.781,Z 340.271,A -85,B 0,C 180,E1 -24622.119,E2 -24622.119} C_VEL
LIN {X 0,Y 138.562,Z 338.134,A -85,B 0,C 180,E1 -24622.737,E2 -24622.737} C_VEL
LIN {X 0,Y 136.702,Z 335.765,A -85,B 0,C 180,E1 -24623.642,E2 -24623.642} C_VEL
LIN {X 0,Y 136.053,Z 333.537,A -85,B 0,C 180,E1 -24624.128,E2 -24624.128} C_VEL
LIN {X 0,Y 136.073,Z 333.532,A -85,B 0,C 180,E1 -24628.903,E2 -24628.903} C_VEL
LIN {X 0,Y 136.156,Z 333.528,A -85,B 0,C 180,E1 -24632.318,E2 -24632.318} C_VEL
LIN {X 0,Y 136.201,Z 333.515,A -85,B 0,C 180,E1 -24638.826,E2 -24638.826} C_VEL
LIN {X 0,Y 136.239,Z 333.474,A -85,B 0,C 180,E1 -24645.053,E2 -24645.053} C_VEL
LIN {X 0,Y 136.439,Z 333.482,A -85,B 0,C 180,E1 -24648.18,E2 -24648.18} C_VEL
LIN {X 0,Y 136.549,Z 333.474,A -85,B 0,C 180,E1 -24651.118,E2 -24651.118} C_VEL
LIN {X 0,Y 137.131,Z 333.353,A -85,B 0,C 180,E1 -24660,E2 -24660} C_VEL
LIN {X 0,Y 136.544,Z 333.465,A -85,B 0,C 180,E1 -24668.883,E2 -24668.883} C_VEL
LIN {X 0,Y 136.426,Z 333.479,A -85,B 0,C 180,E1 -24671.892,E2 -24671.892} C_VEL
LIN {X 0,Y 136.177,Z 333.505,A -85,B 0,C 180,E1 -24678.039,E2 -24678.039} C_VEL
LIN {X 0,Y 136.154,Z 333.519,A -85,B 0,C 180,E1 -24681.686,E2 -24681.686} C_VEL
LIN {X 0,Y 136.047,Z 333.494,A -85,B 0,C 180,E1 -24688.561,E2 -24688.561} C_VEL
LIN {X 0,Y 136.026,Z 333.505,A -85,B 0,C 180,E1 -24694.634,E2 -24694.634} C_VEL
LIN {X 0,Y 136.035,Z 333.539,A -85,B 0,C 180,E1 -24699.189,E2 -24699.189} C_VEL
LIN {X 0,Y 135.988,Z 333.535,A -85,B 0,C 180,E1 -24703.643,E2 -24703.643} C_VEL
LIN {X 0,Y 135.992,Z 333.542,A -85,B 0,C 180,E1 -24707.782,E2 -24707.782} C_VEL
LIN {X 0,Y 136.03,Z 333.541,A -85,B 0,C 180,E1 -24711.676,E2 -24711.676} C_VEL
LIN {X 0,Y 136.062,Z 333.529,A -85,B 0,C 180,E1 -24715.736,E2 -24715.736} C_VEL
LIN {X 0,Y 136.148,Z 333.526,A -85,B 0,C 180,E1 -24722.308,E2 -24722.308} C_VEL
LIN {X 0,Y 136.19,Z 333.529,A -85,B 0,C 180,E1 -24728.635,E2 -24728.635} C_VEL
LIN {X 0,Y 137.101,Z 336.194,A -85,B 0,C 180,E1 -24729.209,E2 -24729.209} C_VEL
LIN {X 0,Y 139.212,Z 338.86,A -85,B 0,C 180,E1 -24730.218,E2 -24730.218} C_VEL
LIN {X 0,Y 141.406,Z 342.214,A -85,B 0,C 180,E1 -24731.274,E2 -24731.274} C_VEL
LIN {X 0,Y 150.362,Z 356.687,A -85,B 0,C 180,E1 -24735.192,E2 -24735.192} C_VEL
LIN {X 0,Y 160.101,Z 375.608,A -85,B 0,C 180,E1 -24739.031,E2 -24739.031} C_VEL
LIN {X 0,Y 162.518,Z 382.181,A -85,B 0,C 180,E1 -24740.001,E2 -24740.001} C_VEL
LIN {X 0,Y 159.043,Z 431.307,A -85,B 0,C 180,E1 -24742.187,E2 -24742.187} C_VEL
LIN {X 0,Y 157.434,Z 444.64,A -85,B 0,C 180,E1 -24743.263,E2 -24743.263} C_VEL
LIN {X 0,Y 155.222,Z 457.47,A -85,B 0,C 180,E1 -24744.796,E2 -24744.796} C_VEL
LIN {X 0,Y 152.58,Z 469.101,A -85,B 0,C 180,E1 -24746.691,E2 -24746.691} C_VEL
LIN {X 0,Y 149.596,Z 479.928,A -85,B 0,C 180,E1 -24748.982,E2 -24748.982} C_VEL
LIN {X 0,Y 146.752,Z 489.273,A -85,B 0,C 180,E1 -24751.512,E2 -24751.512} C_VEL
LIN {X 0,Y 143.548,Z 499.102,A -85,B 0,C 180,E1 -24754.906,E2 -24754.906} C_VEL
LIN {X 0,Y 140.559,Z 507.503,A -85,B 0,C 180,E1 -24758.617,E2 -24758.617} C_VEL
LIN {X 0,Y 138.039,Z 514.818,A -85,B 0,C 180,E1 -24762.744,E2 -24762.744} C_VEL
LIN {X 0,Y 136.292,Z 520.048,A -85,B 0,C 180,E1 -24766.465,E2 -24766.465} C_VEL
LIN {X 0,Y 134.69,Z 525.472,A -85,B 0,C 180,E1 -24771.411,E2 -24771.411} C_VEL
LIN {X 0,Y 133.559,Z 529.575,A -85,B 0,C 180,E1 -24776.548,E2 -24776.548} C_VEL
LIN {X 0,Y 133.108,Z 532.584,A -85,B 0,C 180,E1 -24782.35,E2 -24782.35} C_VEL
LIN {X 0,Y 133.652,Z 534.09,A -85,B 0,C 180,E1 -24787.929,E2 -24787.929} C_VEL
LIN {X 0,Y 135.108,Z 534.271,A -85,B 0,C 180,E1 -24793.26,E2 -24793.26} C_VEL
LIN {X 0,Y 137.35,Z 533.245,A -85,B 0,C 180,E1 -24798.303,E2 -24798.303} C_VEL
LIN {X 0,Y 140.411,Z 531.038,A -85,B 0,C 180,E1 -24803.191,E2 -24803.191} C_VEL
LIN {X 0,Y 144.159,Z 527.829,A -85,B 0,C 180,E1 -24807.57,E2 -24807.57} C_VEL
LIN {X 0,Y 148.784,Z 523.292,A -85,B 0,C 180,E1 -24811.812,E2 -24811.812} C_VEL
LIN {X 0,Y 154.187,Z 517.34,A -85,B 0,C 180,E1 -24815.781,E2 -24815.781} C_VEL
LIN {X 0,Y 160.136,Z 509.83,A -85,B 0,C 180,E1 -24819.445,E2 -24819.445} C_VEL
LIN {X 0,Y 165.483,Z 502.107,A -85,B 0,C 180,E1 -24822.287,E2 -24822.287} C_VEL
LIN {X 0,Y 171.082,Z 492.975,A -85,B 0,C 180,E1 -24824.834,E2 -24824.834} C_VEL
LIN {X 0,Y 176.631,Z 482.384,A -85,B 0,C 180,E1 -24827.068,E2 -24827.068} C_VEL
LIN {X 0,Y 181.331,Z 471.454,A -85,B 0,C 180,E1 -24828.826,E2 -24828.826} C_VEL
LIN {X 0,Y 185.385,Z 459.917,A -85,B 0,C 180,E1 -24830.223,E2 -24830.223} C_VEL
LIN {X 0,Y 188.52,Z 448.249,A -85,B 0,C 180,E1 -24831.306,E2 -24831.306} C_VEL
LIN {X 0,Y 190.992,Z 435.712,A -85,B 0,C 180,E1 -24832.085,E2 -24832.085} C_VEL
LIN {X 0,Y 193.185,Z 417.064,A -85,B 0,C 180,E1 -24832.774,E2 -24832.774} C_VEL
LIN {X 0,Y 194.281,Z 404.744,A -85,B 0,C 180,E1 -24833.262,E2 -24833.262} C_VEL
LIN {X 0,Y 191.186,Z 398.302,A -85,B 0,C 180,E1 -24835.784,E2 -24835.784} C_VEL
LIN {X 0,Y 187.961,Z 392.079,A -85,B 0,C 180,E1 -24838.862,E2 -24838.862} C_VEL
LIN {X 0,Y 186.264,Z 389.19,A -85,B 0,C 180,E1 -24840.7,E2 -24840.7} C_VEL
LIN {X 0,Y 183.859,Z 384.807,A -85,B 0,C 180,E1 -24843.966,E2 -24843.966} C_VEL
LIN {X 0,Y 182.077,Z 381.724,A -85,B 0,C 180,E1 -24847.154,E2 -24847.154} C_VEL
LIN {X 0,Y 180.043,Z 379.837,A -85,B 0,C 180,E1 -24853.545,E2 -24853.545} C_VEL
LIN {X 0,Y 179.934,Z 379.795,A -85,B 0,C 180,E1 -24856.951,E2 -24856.951} C_VEL
LIN {X 0,Y 181.595,Z 381.756,A -85,B 0,C 180,E1 -24863.44,E2 -24863.44} C_VEL
LIN {X 0,Y 182.51,Z 383.716,A -85,B 0,C 180,E1 -24865.503,E2 -24865.503} C_VEL
LIN {X 0,Y 184.781,Z 388.349,A -85,B 0,C 180,E1 -24869.161,E2 -24869.161} C_VEL
LIN {X 0,Y 186.865,Z 392.78,A -85,B 0,C 180,E1 -24871.772,E2 -24871.772} C_VEL
LIN {X 0,Y 188.84,Z 397.387,A -85,B 0,C 180,E1 -24873.935,E2 -24873.935} C_VEL
LIN {X 0,Y 191.334,Z 403.652,A -85,B 0,C 180,E1 -24876.315,E2 -24876.315} C_VEL
LIN {X 0,Y 193.787,Z 410.879,A -85,B 0,C 180,E1 -24878.486,E2 -24878.486} C_VEL
LIN {X 0,Y 193.061,Z 419.41,A -85,B 0,C 180,E1 -24878.843,E2 -24878.843} C_VEL
LIN {X 0,Y 190.667,Z 440.678,A -85,B 0,C 180,E1 -24879.585,E2 -24879.585} C_VEL
LIN {X 0,Y 187.986,Z 454.335,A -85,B 0,C 180,E1 -24880.34,E2 -24880.34} C_VEL
LIN {X 0,Y 184.646,Z 466.088,A -85,B 0,C 180,E1 -24881.275,E2 -24881.275} C_VEL
LIN {X 0,Y 180.234,Z 478.216,A -85,B 0,C 180,E1 -24882.623,E2 -24882.623} C_VEL
LIN {X 0,Y 175.368,Z 489.168,A -85,B 0,C 180,E1 -24884.261,E2 -24884.261} C_VEL
LIN {X 0,Y 170.171,Z 499.135,A -85,B 0,C 180,E1 -24886.244,E2 -24886.244} C_VEL
LIN {X 0,Y 164.651,Z 508.195,A -85,B 0,C 180,E1 -24888.592,E2 -24888.592} C_VEL
LIN {X 0,Y 158.613,Z 517.06,A -85,B 0,C 180,E1 -24891.674,E2 -24891.674} C_VEL
LIN {X 0,Y 153.01,Z 524.285,A -85,B 0,C 180,E1 -24894.974,E2 -24894.974} C_VEL
LIN {X 0,Y 147.575,Z 530.758,A -85,B 0,C 180,E1 -24899.006,E2 -24899.006} C_VEL
LIN {X 0,Y 142.514,Z 536.088,A -85,B 0,C 180,E1 -24903.664,E2 -24903.664} C_VEL
LIN {X 0,Y 140.242,Z 538.392,A -85,B 0,C 180,E1 -24906.377,E2 -24906.377} C_VEL
LIN {X 0,Y 138.194,Z 540.272,A -85,B 0,C 180,E1 -24909.157,E2 -24909.157} C_VEL
LIN {X 0,Y 136.511,Z 541.711,A -85,B 0,C 180,E1 -24912.019,E2 -24912.019} C_VEL
LIN {X 0,Y 134.423,Z 543.459,A -85,B 0,C 180,E1 -24917.939,E2 -24917.939} C_VEL
LIN {X 0,Y 133.822,Z 543.77,A -85,B 0,C 180,E1 -24920.946,E2 -24920.946} C_VEL
LIN {X 0,Y 133.54,Z 543.668,A -85,B 0,C 180,E1 -24923.968,E2 -24923.968} C_VEL
LIN {X 0,Y 133.628,Z 542.491,A -85,B 0,C 180,E1 -24929.4,E2 -24929.4} C_VEL
LIN {X 0,Y 133.42,Z 541.873,A -85,B 0,C 180,E1 -24931.054,E2 -24931.054} C_VEL
LIN {X 0,Y 132.665,Z 541.065,A -85,B 0,C 180,E1 -24932.679,E2 -24932.679} C_VEL
LIN {X 0,Y 130.312,Z 539.109,A -85,B 0,C 180,E1 -24935.873,E2 -24935.873} C_VEL
LIN {X 0,Y 128.022,Z 536.625,A -85,B 0,C 180,E1 -24939.134,E2 -24939.134} C_VEL
LIN {X 0,Y 127.291,Z 534.456,A -85,B 0,C 180,E1 -24941.638,E2 -24941.638} C_VEL
LIN {X 0,Y 127.369,Z 533.679,A -85,B 0,C 180,E1 -24942.474,E2 -24942.474} C_VEL
LIN {X 0,Y 128.885,Z 528.147,A -85,B 0,C 180,E1 -24947.462,E2 -24947.462} C_VEL
LIN {X 0,Y 131.207,Z 521.501,A -85,B 0,C 180,E1 -24952.03,E2 -24952.03} C_VEL
LIN {X 0,Y 133.606,Z 514.851,A -85,B 0,C 180,E1 -24955.652,E2 -24955.652} C_VEL
LIN {X 0,Y 135.942,Z 508.496,A -85,B 0,C 180,E1 -24958.492,E2 -24958.492} C_VEL
LIN {X 0,Y 139.285,Z 498.652,A -85,B 0,C 180,E1 -24962.001,E2 -24962.001} C_VEL
LIN {X 0,Y 142.763,Z 487.974,A -85,B 0,C 180,E1 -24964.918,E2 -24964.918} C_VEL
LIN {X 0,Y 145.817,Z 477.733,A -85,B 0,C 180,E1 -24967.055,E2 -24967.055} C_VEL
LIN {X 0,Y 148.722,Z 465.564,A -85,B 0,C 180,E1 -24968.992,E2 -24968.992} C_VEL
LIN {X 0,Y 151.205,Z 452.232,A -85,B 0,C 180,E1 -24970.494,E2 -24970.494} C_VEL
LIN {X 0,Y 152.943,Z 438.929,A -85,B 0,C 180,E1 -24971.463,E2 -24971.463} C_VEL
LIN {X 0,Y 155.777,Z 398.45,A -85,B 0,C 180,E1 -24973.309,E2 -24973.309} C_VEL
LIN {X 0,Y 154.844,Z 388.95,A -85,B 0,C 180,E1 -24974.136,E2 -24974.136} C_VEL
LIN {X 0,Y 149.163,Z 372.901,A -85,B 0,C 180,E1 -24976.748,E2 -24976.748} C_VEL
LIN {X 0,Y 143.912,Z 360.688,A -85,B 0,C 180,E1 -24979.19,E2 -24979.19} C_VEL
LIN {X 0,Y 139.146,Z 350.777,A -85,B 0,C 180,E1 -24981.556,E2 -24981.556} C_VEL
LIN {X 0,Y 134.106,Z 342.962,A -85,B 0,C 180,E1 -24984.105,E2 -24984.105} C_VEL
LIN {X 0,Y 132.079,Z 339.701,A -85,B 0,C 180,E1 -24985.21,E2 -24985.21} C_VEL
LIN {X 0,Y 129.59,Z 336.527,A -85,B 0,C 180,E1 -24986.57,E2 -24986.57} C_VEL
LIN {X 0,Y 128.978,Z 334.423,A -85,B 0,C 180,E1 -24987.099,E2 -24987.099} C_VEL
LIN {X 0,Y 129.03,Z 334.41,A -85,B 0,C 180,E1 -24990.645,E2 -24990.645} C_VEL
LIN {X 0,Y 129.084,Z 334.406,A -85,B 0,C 180,E1 -24997.772,E2 -24997.772} C_VEL
LIN {X 0,Y 129.16,Z 334.35,A -85,B 0,C 180,E1 -25004.213,E2 -25004.213} C_VEL
LIN {X 0,Y 129.357,Z 334.361,A -85,B 0,C 180,E1 -25007.974,E2 -25007.974} C_VEL
LIN {X 0,Y 129.474,Z 334.357,A -85,B 0,C 180,E1 -25010.628,E2 -25010.628} C_VEL
LIN {X 0,Y 130.086,Z 334.228,A -85,B 0,C 180,E1 -25020,E2 -25020} C_VEL
LIN {X 0,Y 129.471,Z 334.342,A -85,B 0,C 180,E1 -25029.372,E2 -25029.372} C_VEL
LIN {X 0,Y 129.311,Z 334.37,A -85,B 0,C 180,E1 -25032.556,E2 -25032.556} C_VEL
LIN {X 0,Y 129.092,Z 334.385,A -85,B 0,C 180,E1 -25039.066,E2 -25039.066} C_VEL
LIN {X 0,Y 129.045,Z 334.409,A -85,B 0,C 180,E1 -25042.41,E2 -25042.41} C_VEL
LIN {X 0,Y 128.982,Z 334.362,A -85,B 0,C 180,E1 -25049.367,E2 -25049.367} C_VEL
LIN {X 0,Y 128.947,Z 334.392,A -85,B 0,C 180,E1 -25055.148,E2 -25055.148} C_VEL
LIN {X 0,Y 128.933,Z 334.419,A -85,B 0,C 180,E1 -25060.852,E2 -25060.852} C_VEL
LIN {X 0,Y 128.923,Z 334.424,A -85,B 0,C 180,E1 -25065.127,E2 -25065.127} C_VEL
LIN {X 0,Y 128.944,Z 334.412,A -85,B 0,C 180,E1 -25069.735,E2 -25069.735} C_VEL
LIN {X 0,Y 128.966,Z 334.414,A -85,B 0,C 180,E1 -25074.828,E2 -25074.828} C_VEL
LIN {X 0,Y 129.027,Z 334.41,A -85,B 0,C 180,E1 -25080.635,E2 -25080.635} C_VEL
LIN {X 0,Y 129.024,Z 334.413,A -85,B 0,C 180,E1 -25085.611,E2 -25085.611} C_VEL
LIN {X 0,Y 130.024,Z 337.268,A -85,B 0,C 180,E1 -25086.368,E2 -25086.368} C_VEL
LIN {X 0,Y 132.322,Z 339.963,A -85,B 0,C 180,E1 -25087.596,E2 -25087.596} C_VEL
LIN {X 0,Y 134.532,Z 343.252,A -85,B 0,C 180,E1 -25088.772,E2 -25088.772} C_VEL
LIN {X 0,Y 142.038,Z 355.078,A -85,B 0,C 180,E1 -25092.452,E2 -25092.452} C_VEL
LIN {X 0,Y 147.662,Z 364.845,A -85,B 0,C 180,E1 -25094.943,E2 -25094.943} C_VEL
LIN {X 0,Y 155.671,Z 381.234,A -85,B 0,C 180,E1 -25098.255,E2 -25098.255} C_VEL
LIN {X 0,Y 156.576,Z 384.032,A -85,B 0,C 180,E1 -25098.662,E2 -25098.662} C_VEL
LIN {X 0,Y 152.993,Z 431.644,A -85,B 0,C 180,E1 -25100.826,E2 -25100.826} C_VEL
LIN {X 0,Y 151.277,Z 445.391,A -85,B 0,C 180,E1 -25101.98,E2 -25101.98} C_VEL
LIN {X 0,Y 149.207,Z 456.892,A -85,B 0,C 180,E1 -25103.381,E2 -25103.381} C_VEL
LIN {X 0,Y 146.192,Z 469.647,A -85,B 0,C 180,E1 -25105.511,E2 -25105.511} C_VEL
LIN {X 0,Y 143.099,Z 480.418,A -85,B 0,C 180,E1 -25107.88,E2 -25107.88} C_VEL
LIN {X 0,Y 139.987,Z 490.158,A -85,B 0,C 180,E1 -25110.637,E2 -25110.637} C_VEL
LIN {X 0,Y 137.093,Z 498.61,A -85,B 0,C 180,E1 -25113.664,E2 -25113.664} C_VEL
LIN {X 0,Y 133.731,Z 507.712,A -85,B 0,C 180,E1 -25117.826,E2 -25117.826} C_VEL
LIN {X 0,Y 130.955,Z 515.389,A -85,B 0,C 180,E1 -25122.385,E2 -25122.385} C_VEL
LIN {X 0,Y 128.738,Z 521.904,A -85,B 0,C 180,E1 -25127.461,E2 -25127.461} C_VEL
LIN {X 0,Y 127.21,Z 526.945,A -85,B 0,C 180,E1 -25132.738,E2 -25132.738} C_VEL
LIN {X 0,Y 126.344,Z 530.072,A -85,B 0,C 180,E1 -25137.125,E2 -25137.125} C_VEL
LIN {X 0,Y 126.037,Z 532.988,A -85,B 0,C 180,E1 -25143.235,E2 -25143.235} C_VEL
LIN {X 0,Y 126.755,Z 534.417,A -85,B 0,C 180,E1 -25149.082,E2 -25149.082} C_VEL
LIN {X 0,Y 128.682,Z 534.45,A -85,B 0,C 180,E1 -25155.217,E2 -25155.217} C_VEL
LIN {X 0,Y 130.987,Z 533.447,A -85,B 0,C 180,E1 -25159.92,E2 -25159.92} C_VEL
LIN {X 0,Y 134.277,Z 531.277,A -85,B 0,C 180,E1 -25164.849,E2 -25164.849} C_VEL
LIN {X 0,Y 138.544,Z 527.891,A -85,B 0,C 180,E1 -25169.558,E2 -25169.558} C_VEL
LIN {X 0,Y 143.515,Z 523.358,A -85,B 0,C 180,E1 -25173.849,E2 -25173.849} C_VEL
LIN {X 0,Y 149.366,Z 517.335,A -85,B 0,C 180,E1 -25177.888,E2 -25177.888} C_VEL
LIN {X 0,Y 155.581,Z 509.869,A -85,B 0,C 180,E1 -25181.516,E2 -25181.516} C_VEL
LIN {X 0,Y 162.034,Z 500.91,A -85,B 0,C 180,E1 -25184.739,E2 -25184.739} C_VEL
LIN {X 0,Y 167.463,Z 492.324,A -85,B 0,C 180,E1 -25187.03,E2 -25187.03} C_VEL
LIN {X 0,Y 172.679,Z 482.728,A -85,B 0,C 180,E1 -25189.016,E2 -25189.016} C_VEL
LIN {X 0,Y 177.359,Z 472.426,A -85,B 0,C 180,E1 -25190.672,E2 -25190.672} C_VEL
LIN {X 0,Y 181.539,Z 461.186,A -85,B 0,C 180,E1 -25192.048,E2 -25192.048} C_VEL
LIN {X 0,Y 185.17,Z 448.391,A -85,B 0,C 180,E1 -25193.235,E2 -25193.235} C_VEL
LIN {X 0,Y 187.802,Z 435.395,A -85,B 0,C 180,E1 -25194.009,E2 -25194.009} C_VEL
LIN {X 0,Y 190.224,Z 414.756,A -85,B 0,C 180,E1 -25194.758,E2 -25194.758} C_VEL
LIN {X 0,Y 190.817,Z 408.435,A -85,B 0,C 180,E1 -25195.005,E2 -25195.005} C_VEL
LIN {X 0,Y 188.265,Z 402.929,A -85,B 0,C 180,E1 -25197.337,E2 -25197.337} C_VEL
LIN {X 0,Y 185.66,Z 397.665,A -85,B 0,C 180,E1 -25200.105,E2 -25200.105} C_VEL
LIN {X 0,Y 183.965,Z 394.679,A -85,B 0,C 180,E1 -25202.189,E2 -25202.189} C_VEL
LIN {X 0,Y 182.342,Z 391.426,A -85,B 0,C 180,E1 -25204.656,E2 -25204.656} C_VEL
LIN {X 0,Y 180.78,Z 388.588,A -85,B 0,C 180,E1 -25207.713,E2 -25207.713} C_VEL
LIN {X 0,Y 179.035,Z 386.853,A -85,B 0,C 180,E1 -25213.623,E2 -25213.623} C_VEL
LIN {X 0,Y 178.942,Z 386.852,A -85,B 0,C 180,E1 -25217.048,E2 -25217.048} C_VEL
LIN {X 0,Y 180.427,Z 388.686,A -85,B 0,C 180,E1 -25223.093,E2 -25223.093} C_VEL
LIN {X 0,Y 181.501,Z 391.406,A -85,B 0,C 180,E1 -25225.655,E2 -25225.655} C_VEL
LIN {X 0,Y 183.108,Z 394.676,A -85,B 0,C 180,E1 -25228.326,E2 -25228.326} C_VEL
LIN {X 0,Y 184.983,Z 399.073,A -85,B 0,C 180,E1 -25230.937,E2 -25230.937} C_VEL
LIN {X 0,Y 187.152,Z 404.561,A -85,B 0,C 180,E1 -25233.47,E2 -25233.47} C_VEL
LIN {X 0,Y 189.152,Z 410.245,A -85,B 0,C 180,E1 -25235.558,E2 -25235.558} C_VEL
LIN {X 0,Y 190.396,Z 414.027,A -85,B 0,C 180,E1 -25236.746,E2 -25236.746} C_VEL
LIN {X 0,Y 187.557,Z 439.576,A -85,B 0,C 180,E1 -25237.634,E2 -25237.634} C_VEL
LIN {X 0,Y 184.726,Z 453.654,A -85,B 0,C 180,E1 -25238.382,E2 -25238.382} C_VEL
LIN {X 0,Y 181.458,Z 464.959,A -85,B 0,C 180,E1 -25239.246,E2 -25239.246} C_VEL
LIN {X 0,Y 177.536,Z 475.679,A -85,B 0,C 180,E1 -25240.372,E2 -25240.372} C_VEL
LIN {X 0,Y 172.392,Z 487.012,A -85,B 0,C 180,E1 -25241.942,E2 -25241.942} C_VEL
LIN {X 0,Y 166.357,Z 498.339,A -85,B 0,C 180,E1 -25244.11,E2 -25244.11} C_VEL
LIN {X 0,Y 160.598,Z 507.502,A -85,B 0,C 180,E1 -25246.445,E2 -25246.445} C_VEL
LIN {X 0,Y 156.217,Z 513.683,A -85,B 0,C 180,E1 -25248.441,E2 -25248.441} C_VEL
LIN {X 0,Y 150.157,Z 521.485,A -85,B 0,C 180,E1 -25251.687,E2 -25251.687} C_VEL
LIN {X 0,Y 145.451,Z 526.82,A -85,B 0,C 180,E1 -25254.576,E2 -25254.576} C_VEL
LIN {X 0,Y 140.175,Z 532.484,A -85,B 0,C 180,E1 -25258.673,E2 -25258.673} C_VEL
LIN {X 0,Y 134.906,Z 537.4,A -85,B 0,C 180,E1 -25263.729,E2 -25263.729} C_VEL
LIN {X 0,Y 131.562,Z 540.254,A -85,B 0,C 180,E1 -25268.054,E2 -25268.054} C_VEL
LIN {X 0,Y 129.745,Z 541.635,A -85,B 0,C 180,E1 -25271.046,E2 -25271.046} C_VEL
LIN {X 0,Y 127.452,Z 543.27,A -85,B 0,C 180,E1 -25277.269,E2 -25277.269} C_VEL
LIN {X 0,Y 126.474,Z 543.324,A -85,B 0,C 180,E1 -25283.63,E2 -25283.63} C_VEL
LIN {X 0,Y 126.563,Z 542.01,A -85,B 0,C 180,E1 -25289.486,E2 -25289.486} C_VEL
LIN {X 0,Y 126.495,Z 540.439,A -85,B 0,C 180,E1 -25293.195,E2 -25293.195} C_VEL
LIN {X 0,Y 126.683,Z 537.481,A -85,B 0,C 180,E1 -25297.982,E2 -25297.982} C_VEL
LIN {X 0,Y 127.369,Z 533.679,A -85,B 0,C 180,E1 -25302.474,E2 -25302.474} C_VEL
LIN {X 0,Y 127.314,Z 531.259,A -85,B 0,C 180,E1 -25304.903,E2 -25304.903} C_VEL
LIN {X 0,Y 125.837,Z 526.661,A -85,B 0,C 180,E1 -25308.835,E2 -25308.835} C_VEL
LIN {X 0,Y 124.849,Z 521.359,A -85,B 0,C 180,E1 -25312.661,E2 -25312.661} C_VEL
LIN {X 0,Y 125.549,Z 517.833,A -85,B 0,C 180,E1 -25314.82,E2 -25314.82} C_VEL
LIN {X 0,Y 128.585,Z 509.851,A -85,B 0,C 180,E1 -25318.832,E2 -25318.832} C_VEL
LIN {X 0,Y 132.119,Z 500.231,A -85,B 0,C 180,E1 -25322.597,E2 -25322.597} C_VEL
LIN {X 0,Y 135.648,Z 489.942,A -85,B 0,C 180,E1 -25325.662,E2 -25325.662} C_VEL
LIN {X 0,Y 139.28,Z 478.63,A -85,B 0,C 180,E1 -25328.188,E2 -25328.188} C_VEL
LIN {X 0,Y 142.282,Z 466.886,A -85,B 0,C 180,E1 -25330.191,E2 -25330.191} C_VEL
LIN {X 0,Y 144.837,Z 454.126,A -85,B 0,C 180,E1 -25331.743,E2 -25331.743} C_VEL
LIN {X 0,Y 146.813,Z 440.679,A -85,B 0,C 180,E1 -25332.818,E2 -25332.818} C_VEL
LIN {X 0,Y 149.886,Z 399.325,A -85,B 0,C 180,E1 -25334.789,E2 -25334.789} C_VEL
LIN {X 0,Y 149.294,Z 391.694,A -85,B 0,C 180,E1 -25335.455,E2 -25335.455} C_VEL
LIN {X 0,Y 144.017,Z 376.511,A -85,B 0,C 180,E1 -25338.031,E2 -25338.031} C_VEL
LIN {X 0,Y 139.258,Z 365.094,A -85,B 0,C 180,E1 -25340.43,E2 -25340.43} C_VEL
LIN {X 0,Y 134.578,Z 355.194,A -85,B 0,C 180,E1 -25342.929,E2 -25342.929} C_VEL
LIN {X 0,Y 129.722,Z 347.606,A -85,B 0,C 180,E1 -25345.54,E2 -25345.54} C_VEL
LIN {X 0,Y 127.424,Z 344.104,A -85,B 0,C 180,E1 -25346.881,E2 -25346.881} C_VEL
LIN {X 0,Y 125.322,Z 340.956,A -85,B 0,C 180,E1 -25348.164,E2 -25348.164} C_VEL
LIN {X 0,Y 124.395,Z 339.752,A -85,B 0,C 180,E1 -25348.73,E2 -25348.73} C_VEL
LIN {X 0,Y 122.604,Z 337.441,A -85,B 0,C 180,E1 -25349.867,E2 -25349.867} C_VEL
LIN {X 0,Y 121.981,Z 335.287,A -85,B 0,C 180,E1 -25350.425,E2 -25350.425} C_VEL
LIN {X 0,Y 122.018,Z 335.286,A -85,B 0,C 180,E1 -25357.175,E2 -25357.175} C_VEL
LIN {X 0,Y 122.073,Z 335.23,A -85,B 0,C 180,E1 -25363.27,E2 -25363.27} C_VEL
LIN {X 0,Y 122.3,Z 335.237,A -85,B 0,C 180,E1 -25367.695,E2 -25367.695} C_VEL
LIN {X 0,Y 122.403,Z 335.237,A -85,B 0,C 180,E1 -25370.081,E2 -25370.081} C_VEL
LIN {X 0,Y 122.578,Z 335.153,A -85,B 0,C 180,E1 -25376.713,E2 -25376.713} C_VEL
LIN {X 0,Y 123.039,Z 335.103,A -85,B 0,C 180,E1 -25380,E2 -25380} C_VEL
LIN {X 0,Y 122.405,Z 335.234,A -85,B 0,C 180,E1 -25386.803,E2 -25386.803} C_VEL
LIN {X 0,Y 122.3,Z 335.24,A -85,B 0,C 180,E1 -25392.304,E2 -25392.304} C_VEL
LIN {X 0,Y 122.071,Z 335.271,A -85,B 0,C 180,E1 -25396.73,E2 -25396.73} C_VEL
LIN {X 0,Y 121.964,Z 335.291,A -85,B 0,C 180,E1 -25402.765,E2 -25402.765} C_VEL
LIN {X 0,Y 121.906,Z 335.235,A -85,B 0,C 180,E1 -25410.13,E2 -25410.13} C_VEL
LIN {X 0,Y 121.878,Z 335.283,A -85,B 0,C 180,E1 -25416.155,E2 -25416.155} C_VEL
LIN {X 0,Y 121.857,Z 335.297,A -85,B 0,C 180,E1 -25421.418,E2 -25421.418} C_VEL
LIN {X 0,Y 121.873,Z 335.294,A -85,B 0,C 180,E1 -25428.562,E2 -25428.562} C_VEL
LIN {X 0,Y 121.917,Z 335.292,A -85,B 0,C 180,E1 -25434.788,E2 -25434.788} C_VEL
LIN {X 0,Y 121.952,Z 335.291,A -85,B 0,C 180,E1 -25441.195,E2 -25441.195} C_VEL
LIN {X 0,Y 121.938,Z 335.295,A -85,B 0,C 180,E1 -25442.199,E2 -25442.199} C_VEL
LIN {X 0,Y 122.848,Z 337.998,A -85,B 0,C 180,E1 -25442.972,E2 -25442.972} C_VEL
LIN {X 0,Y 125.03,Z 340.291,A -85,B 0,C 180,E1 -25444.291,E2 -25444.291} C_VEL
LIN {X 0,Y 127.353,Z 344.021,A -85,B 0,C 180,E1 -25445.751,E2 -25445.751} C_VEL
LIN {X 0,Y 128.652,Z 345.695,A -85,B 0,C 180,E1 -25446.495,E2 -25446.495} C_VEL
LIN {X 0,Y 133.688,Z 353.48,A -85,B 0,C 180,E1 -25449.27,E2 -25449.27} C_VEL
LIN {X 0,Y 140.878,Z 365.349,A -85,B 0,C 180,E1 -25452.813,E2 -25452.813} C_VEL
LIN {X 0,Y 150.006,Z 383.691,A -85,B 0,C 180,E1 -25456.878,E2 -25456.878} C_VEL
LIN {X 0,Y 150.703,Z 386.077,A -85,B 0,C 180,E1 -25457.23,E2 -25457.23} C_VEL
LIN {X 0,Y 147.091,Z 431.51,A -85,B 0,C 180,E1 -25459.322,E2 -25459.322} C_VEL
LIN {X 0,Y 145.283,Z 445.411,A -85,B 0,C 180,E1 -25460.507,E2 -25460.507} C_VEL
LIN {X 0,Y 143.053,Z 457.312,A -85,B 0,C 180,E1 -25461.996,E2 -25461.996} C_VEL
LIN {X 0,Y 139.884,Z 470.174,A -85,B 0,C 180,E1 -25464.224,E2 -25464.224} C_VEL
LIN {X 0,Y 136.658,Z 480.889,A -85,B 0,C 180,E1 -25466.674,E2 -25466.674} C_VEL
LIN {X 0,Y 132.938,Z 491.89,A -85,B 0,C 180,E1 -25469.99,E2 -25469.99} C_VEL
LIN {X 0,Y 129.335,Z 501.715,A -85,B 0,C 180,E1 -25473.884,E2 -25473.884} C_VEL
LIN {X 0,Y 126.243,Z 509.755,A -85,B 0,C 180,E1 -25477.988,E2 -25477.988} C_VEL
LIN {X 0,Y 123.308,Z 517.489,A -85,B 0,C 180,E1 -25483.166,E2 -25483.166} C_VEL
LIN {X 0,Y 121.188,Z 523.604,A -85,B 0,C 180,E1 -25488.587,E2 -25488.587} C_VEL
LIN {X 0,Y 119.764,Z 528.336,A -85,B 0,C 180,E1 -25494.24,E2 -25494.24} C_VEL
LIN {X 0,Y 119.088,Z 530.751,A -85,B 0,C 180,E1 -25498.158,E2 -25498.158} C_VEL
LIN {X 0,Y 118.985,Z 533.377,A -85,B 0,C 180,E1 -25504.215,E2 -25504.215} C_VEL
LIN {X 0,Y 119.92,Z 534.732,A -85,B 0,C 180,E1 -25510.37,E2 -25510.37} C_VEL
LIN {X 0,Y 121.882,Z 534.771,A -85,B 0,C 180,E1 -25516.215,E2 -25516.215} C_VEL
LIN {X 0,Y 124.88,Z 533.567,A -85,B 0,C 180,E1 -25521.967,E2 -25521.967} C_VEL
LIN {X 0,Y 128.375,Z 531.458,A -85,B 0,C 180,E1 -25526.807,E2 -25526.807} C_VEL
LIN {X 0,Y 133.003,Z 528.08,A -85,B 0,C 180,E1 -25531.604,E2 -25531.604} C_VEL
LIN {X 0,Y 138.488,Z 523.425,A -85,B 0,C 180,E1 -25536.047,E2 -25536.047} C_VEL
LIN {X 0,Y 144.706,Z 517.349,A -85,B 0,C 180,E1 -25540.125,E2 -25540.125} C_VEL
LIN {X 0,Y 151.511,Z 509.602,A -85,B 0,C 180,E1 -25543.84,E2 -25543.84} C_VEL
LIN {X 0,Y 157.153,Z 502.21,A -85,B 0,C 180,E1 -25546.523,E2 -25546.523} C_VEL
LIN {X 0,Y 163.59,Z 492.637,A -85,B 0,C 180,E1 -25549.11,E2 -25549.11} C_VEL
LIN {X 0,Y 169.295,Z 482.478,A -85,B 0,C 180,E1 -25551.177,E2 -25551.177} C_VEL
LIN {X 0,Y 174.311,Z 471.741,A -85,B 0,C 180,E1 -25552.838,E2 -25552.838} C_VEL
LIN {X 0,Y 178.772,Z 459.936,A -85,B 0,C 180,E1 -25554.212,E2 -25554.212} C_VEL
LIN {X 0,Y 182.417,Z 446.936,A -85,B 0,C 180,E1 -25555.338,E2 -25555.338} C_VEL
LIN {X 0,Y 184.998,Z 434.09,A -85,B 0,C 180,E1 -25556.041,E2 -25556.041} C_VEL
LIN {X 0,Y 187.537,Z 412.095,A -85,B 0,C 180,E1 -25556.839,E2 -25556.839} C_VEL
LIN {X 0,Y 184.328,Z 404.976,A -85,B 0,C 180,E1 -25560.318,E2 -25560.318} C_VEL
LIN {X 0,Y 182.77,Z 401.924,A -85,B 0,C 180,E1 -25562.328,E2 -25562.328} C_VEL
LIN {X 0,Y 180.843,Z 398.015,A -85,B 0,C 180,E1 -25565.377,E2 -25565.377} C_VEL
LIN {X 0,Y 179.607,Z 395.538,A -85,B 0,C 180,E1 -25568.046,E2 -25568.046} C_VEL
LIN {X 0,Y 178.025,Z 393.88,A -85,B 0,C 180,E1 -25573.702,E2 -25573.702} C_VEL
LIN {X 0,Y 177.951,Z 393.901,A -85,B 0,C 180,E1 -25577.146,E2 -25577.146} C_VEL
LIN {X 0,Y 179.283,Z 395.648,A -85,B 0,C 180,E1 -25582.791,E2 -25582.791} C_VEL
LIN {X 0,Y 181.416,Z 400.869,A -85,B 0,C 180,E1 -25587.378,E2 -25587.378} C_VEL
LIN {X 0,Y 183.086,Z 405.221,A -85,B 0,C 180,E1 -25590.002,E2 -25590.002} C_VEL
LIN {X 0,Y 185.229,Z 411.032,A -85,B 0,C 180,E1 -25592.707,E2 -25592.707} C_VEL
LIN {X 0,Y 187.077,Z 417.153,A -85,B 0,C 180,E1 -25594.867,E2 -25594.867} C_VEL
LIN {X 0,Y 184.58,Z 439.046,A -85,B 0,C 180,E1 -25595.643,E2 -25595.643} C_VEL
LIN {X 0,Y 181.887,Z 452.296,A -85,B 0,C 180,E1 -25596.321,E2 -25596.321} C_VEL
LIN {X 0,Y 178.357,Z 464.354,A -85,B 0,C 180,E1 -25597.192,E2 -25597.192} C_VEL
LIN {X 0,Y 173.762,Z 476.351,A -85,B 0,C 180,E1 -25598.422,E2 -25598.422} C_VEL
LIN {X 0,Y 168.442,Z 487.52,A -85,B 0,C 180,E1 -25599.961,E2 -25599.961} C_VEL
LIN {X 0,Y 162.807,Z 497.641,A -85,B 0,C 180,E1 -25601.888,E2 -25601.888} C_VEL
LIN {X 0,Y 156.786,Z 506.858,A -85,B 0,C 180,E1 -25604.192,E2 -25604.192} C_VEL
LIN {X 0,Y 151.024,Z 514.501,A -85,B 0,C 180,E1 -25606.67,E2 -25606.67} C_VEL
LIN {X 0,Y 144.672,Z 522.049,A -85,B 0,C 180,E1 -25609.949,E2 -25609.949} C_VEL
LIN {X 0,Y 137.917,Z 529.099,A -85,B 0,C 180,E1 -25614.14,E2 -25614.14} C_VEL
LIN {X 0,Y 132.97,Z 533.833,A -85,B 0,C 180,E1 -25618.107,E2 -25618.107} C_VEL
LIN {X 0,Y 128.556,Z 537.516,A -85,B 0,C 180,E1 -25622.324,E2 -25622.324} C_VEL
LIN {X 0,Y 124.986,Z 540.238,A -85,B 0,C 180,E1 -25626.834,E2 -25626.834} C_VEL
LIN {X 0,Y 121.571,Z 542.508,A -85,B 0,C 180,E1 -25633.211,E2 -25633.211} C_VEL
LIN {X 0,Y 119.781,Z 543.196,A -85,B 0,C 180,E1 -25639.874,E2 -25639.874} C_VEL
LIN {X 0,Y 119.351,Z 542.372,A -85,B 0,C 180,E1 -25646.635,E2 -25646.635} C_VEL
LIN {X 0,Y 119.487,Z 541.059,A -85,B 0,C 180,E1 -25650.768,E2 -25650.768} C_VEL
LIN {X 0,Y 119.515,Z 537.948,A -85,B 0,C 180,E1 -25656.765,E2 -25656.765} C_VEL
LIN {X 0,Y 120.125,Z 534.15,A -85,B 0,C 180,E1 -25661.826,E2 -25661.826} C_VEL
LIN {X 0,Y 121.466,Z 529.18,A -85,B 0,C 180,E1 -25666.826,E2 -25666.826} C_VEL
LIN {X 0,Y 123.719,Z 522.904,A -85,B 0,C 180,E1 -25671.678,E2 -25671.678} C_VEL
LIN {X 0,Y 125.549,Z 517.833,A -85,B 0,C 180,E1 -25674.82,E2 -25674.82} C_VEL
LIN {X 0,Y 126.365,Z 514.157,A -85,B 0,C 180,E1 -25676.873,E2 -25676.873} C_VEL
LIN {X 0,Y 126.155,Z 507.667,A -85,B 0,C 180,E1 -25680.266,E2 -25680.266} C_VEL
LIN {X 0,Y 126.107,Z 500.642,A -85,B 0,C 180,E1 -25683.469,E2 -25683.469} C_VEL
LIN {X 0,Y 127.136,Z 496.088,A -85,B 0,C 180,E1 -25685.137,E2 -25685.137} C_VEL
LIN {X 0,Y 130.883,Z 485.27,A -85,B 0,C 180,E1 -25688.144,E2 -25688.144} C_VEL
LIN {X 0,Y 134.143,Z 474.418,A -85,B 0,C 180,E1 -25690.427,E2 -25690.427} C_VEL
LIN {X 0,Y 137.146,Z 462.568,A -85,B 0,C 180,E1 -25692.276,E2 -25692.276} C_VEL
LIN {X 0,Y 139.609,Z 449.875,A -85,B 0,C 180,E1 -25693.688,E2 -25693.688} C_VEL
LIN {X 0,Y 141.359,Z 436.198,A -85,B 0,C 180,E1 -25694.647,E2 -25694.647} C_VEL
LIN {X 0,Y 144.109,Z 399.338,A -85,B 0,C 180,E1 -25696.418,E2 -25696.418} C_VEL
LIN {X 0,Y 143.555,Z 393.655,A -85,B 0,C 180,E1 -25696.974,E2 -25696.974} C_VEL
LIN {X 0,Y 138.357,Z 378.539,A -85,B 0,C 180,E1 -25699.729,E2 -25699.729} C_VEL
LIN {X 0,Y 133.754,Z 367.44,A -85,B 0,C 180,E1 -25702.261,E2 -25702.261} C_VEL
LIN {X 0,Y 129.967,Z 359.462,A -85,B 0,C 180,E1 -25704.417,E2 -25704.417} C_VEL
LIN {X 0,Y 125.117,Z 351.693,A -85,B 0,C 180,E1 -25707.272,E2 -25707.272} C_VEL
LIN {X 0,Y 120.92,Z 345.384,A -85,B 0,C 180,E1 -25709.984,E2 -25709.984} C_VEL
LIN {X 0,Y 118.728,Z 342.295,A -85,B 0,C 180,E1 -25711.501,E2 -25711.501} C_VEL
LIN {X 0,Y 118.005,Z 341.205,A -85,B 0,C 180,E1 -25712.03,E2 -25712.03} C_VEL
LIN {X 0,Y 115.755,Z 338.858,A -85,B 0,C 180,E1 -25713.642,E2 -25713.642} C_VEL
LIN {X 0,Y 114.863,Z 336.168,A -85,B 0,C 180,E1 -25714.64,E2 -25714.64} C_VEL
LIN {X 0,Y 114.959,Z 336.162,A -85,B 0,C 180,E1 -25718.481,E2 -25718.481} C_VEL
LIN {X 0,Y 115.093,Z 336.109,A -85,B 0,C 180,E1 -25725.862,E2 -25725.862} C_VEL
LIN {X 0,Y 115.318,Z 336.119,A -85,B 0,C 180,E1 -25729.465,E2 -25729.465} C_VEL
LIN {X 0,Y 115.504,Z 336.033,A -85,B 0,C 180,E1 -25736.512,E2 -25736.512} C_VEL
LIN {X 0,Y 115.99,Z 335.978,A -85,B 0,C 180,E1 -25740,E2 -25740} C_VEL
LIN {X 0,Y 115.36,Z 336.114,A -85,B 0,C 180,E1 -25746.999,E2 -25746.999} C_VEL
LIN {X 0,Y 115.217,Z 336.124,A -85,B 0,C 180,E1 -25752.553,E2 -25752.553} C_VEL
LIN {X 0,Y 114.976,Z 336.146,A -85,B 0,C 180,E1 -25757.796,E2 -25757.796} C_VEL
LIN {X 0,Y 114.891,Z 336.172,A -85,B 0,C 180,E1 -25763.407,E2 -25763.407} C_VEL
LIN {X 0,Y 114.837,Z 336.11,A -85,B 0,C 180,E1 -25771.026,E2 -25771.026} C_VEL
LIN {X 0,Y 114.78,Z 336.183,A -85,B 0,C 180,E1 -25777.756,E2 -25777.756} C_VEL
LIN {X 0,Y 114.771,Z 336.175,A -85,B 0,C 180,E1 -25782.695,E2 -25782.695} C_VEL
LIN {X 0,Y 114.797,Z 336.181,A -85,B 0,C 180,E1 -25787.655,E2 -25787.655} C_VEL
LIN {X 0,Y 114.794,Z 336.189,A -85,B 0,C 180,E1 -25792.74,E2 -25792.74} C_VEL
LIN {X 0,Y 114.853,Z 336.289,A -85,B 0,C 180,E1 -25798.163,E2 -25798.163} C_VEL
LIN {X 0,Y 115.792,Z 338.902,A -85,B 0,C 180,E1 -25799.056,E2 -25799.056} C_VEL
LIN {X 0,Y 118.093,Z 341.26,A -85,B 0,C 180,E1 -25800.704,E2 -25800.704} C_VEL
LIN {X 0,Y 120.377,Z 344.888,A -85,B 0,C 180,E1 -25802.356,E2 -25802.356} C_VEL
LIN {X 0,Y 121.93,Z 346.895,A -85,B 0,C 180,E1 -25803.37,E2 -25803.37} C_VEL
LIN {X 0,Y 125.455,Z 352.044,A -85,B 0,C 180,E1 -25805.59,E2 -25805.59} C_VEL
LIN {X 0,Y 129.651,Z 358.63,A -85,B 0,C 180,E1 -25808.055,E2 -25808.055} C_VEL
LIN {X 0,Y 136.403,Z 370.055,A -85,B 0,C 180,E1 -25811.596,E2 -25811.596} C_VEL
LIN {X 0,Y 144.761,Z 387.206,A -85,B 0,C 180,E1 -25815.609,E2 -25815.609} C_VEL
LIN {X 0,Y 141.155,Z 432.189,A -85,B 0,C 180,E1 -25817.785,E2 -25817.785} C_VEL
LIN {X 0,Y 139.388,Z 445.099,A -85,B 0,C 180,E1 -25818.908,E2 -25818.908} C_VEL
LIN {X 0,Y 136.878,Z 458.013,A -85,B 0,C 180,E1 -25820.571,E2 -25820.571} C_VEL
LIN {X 0,Y 133.68,Z 470.346,A -85,B 0,C 180,E1 -25822.775,E2 -25822.775} C_VEL
LIN {X 0,Y 130.281,Z 481.225,A -85,B 0,C 180,E1 -25825.349,E2 -25825.349} C_VEL
LIN {X 0,Y 126.54,Z 491.822,A -85,B 0,C 180,E1 -25828.653,E2 -25828.653} C_VEL
LIN {X 0,Y 122.965,Z 501.129,A -85,B 0,C 180,E1 -25832.446,E2 -25832.446} C_VEL
LIN {X 0,Y 119.672,Z 509.311,A -85,B 0,C 180,E1 -25836.734,E2 -25836.734} C_VEL
LIN {X 0,Y 117.012,Z 515.94,A -85,B 0,C 180,E1 -25841.177,E2 -25841.177} C_VEL
LIN {X 0,Y 114.905,Z 521.546,A -85,B 0,C 180,E1 -25845.963,E2 -25845.963} C_VEL
LIN {X 0,Y 113.128,Z 526.831,A -85,B 0,C 180,E1 -25851.871,E2 -25851.871} C_VEL
LIN {X 0,Y 112.309,Z 529.597,A -85,B 0,C 180,E1 -25855.964,E2 -25855.964} C_VEL
LIN {X 0,Y 111.83,Z 531.839,A -85,B 0,C 180,E1 -25860.167,E2 -25860.167} C_VEL
LIN {X 0,Y 111.98,Z 533.769,A -85,B 0,C 180,E1 -25865.323,E2 -25865.323} C_VEL
LIN {X 0,Y 113.15,Z 535.031,A -85,B 0,C 180,E1 -25871.811,E2 -25871.811} C_VEL
LIN {X 0,Y 115.376,Z 535.028,A -85,B 0,C 180,E1 -25877.928,E2 -25877.928} C_VEL
LIN {X 0,Y 118.557,Z 533.887,A -85,B 0,C 180,E1 -25883.644,E2 -25883.644} C_VEL
LIN {X 0,Y 122.806,Z 531.554,A -85,B 0,C 180,E1 -25889.113,E2 -25889.113} C_VEL
LIN {X 0,Y 127.777,Z 528.197,A -85,B 0,C 180,E1 -25893.895,E2 -25893.895} C_VEL
LIN {X 0,Y 133.684,Z 523.508,A -85,B 0,C 180,E1 -25898.407,E2 -25898.407} C_VEL
LIN {X 0,Y 140.293,Z 517.404,A -85,B 0,C 180,E1 -25902.508,E2 -25902.508} C_VEL
LIN {X 0,Y 147.594,Z 509.55,A -85,B 0,C 180,E1 -25906.226,E2 -25906.226} C_VEL
LIN {X 0,Y 154.656,Z 500.618,A -85,B 0,C 180,E1 -25909.325,E2 -25909.325} C_VEL
LIN {X 0,Y 160.713,Z 491.711,A -85,B 0,C 180,E1 -25911.565,E2 -25911.565} C_VEL
LIN {X 0,Y 167.027,Z 480.625,A -85,B 0,C 180,E1 -25913.689,E2 -25913.689} C_VEL
LIN {X 0,Y 172.33,Z 469.275,A -85,B 0,C 180,E1 -25915.321,E2 -25915.321} C_VEL
LIN {X 0,Y 177.124,Z 456.098,A -85,B 0,C 180,E1 -25916.686,E2 -25916.686} C_VEL
LIN {X 0,Y 180.472,Z 443.618,A -85,B 0,C 180,E1 -25917.629,E2 -25917.629} C_VEL
LIN {X 0,Y 182.889,Z 430.327,A -85,B 0,C 180,E1 -25918.229,E2 -25918.229} C_VEL
LIN {X 0,Y 184.516,Z 416.137,A -85,B 0,C 180,E1 -25918.713,E2 -25918.713} C_VEL
LIN {X 0,Y 182.124,Z 410.468,A -85,B 0,C 180,E1 -25921.671,E2 -25921.671} C_VEL
LIN {X 0,Y 179.417,Z 404.626,A -85,B 0,C 180,E1 -25926.073,E2 -25926.073} C_VEL
LIN {X 0,Y 178.44,Z 402.486,A -85,B 0,C 180,E1 -25928.383,E2 -25928.383} C_VEL
LIN {X 0,Y 177.016,Z 400.904,A -85,B 0,C 180,E1 -25933.781,E2 -25933.781} C_VEL
LIN {X 0,Y 177,Z 401.033,A -85,B 0,C 180,E1 -25937.683,E2 -25937.683} C_VEL
LIN {X 0,Y 178.145,Z 402.569,A -85,B 0,C 180,E1 -25942.474,E2 -25942.474} C_VEL
LIN {X 0,Y 179.942,Z 407.653,A -85,B 0,C 180,E1 -25946.756,E2 -25946.756} C_VEL
LIN {X 0,Y 181.258,Z 411.306,A -85,B 0,C 180,E1 -25948.998,E2 -25948.998} C_VEL
LIN {X 0,Y 183.126,Z 416.966,A -85,B 0,C 180,E1 -25951.672,E2 -25951.672} C_VEL
LIN {X 0,Y 184.119,Z 420.486,A -85,B 0,C 180,E1 -25952.968,E2 -25952.968} C_VEL
LIN {X 0,Y 181.63,Z 440.181,A -85,B 0,C 180,E1 -25953.645,E2 -25953.645} C_VEL
LIN {X 0,Y 178.675,Z 453.58,A -85,B 0,C 180,E1 -25954.328,E2 -25954.328} C_VEL
LIN {X 0,Y 174.395,Z 466.859,A -85,B 0,C 180,E1 -25955.326,E2 -25955.326} C_VEL
LIN {X 0,Y 169.525,Z 478.58,A -85,B 0,C 180,E1 -25956.579,E2 -25956.579} C_VEL
LIN {X 0,Y 164.059,Z 489.26,A -85,B 0,C 180,E1 -25958.098,E2 -25958.098} C_VEL
LIN {X 0,Y 158.218,Z 498.983,A -85,B 0,C 180,E1 -25960,E2 -25960} C_VEL
LIN {X 0,Y 151.979,Z 507.891,A -85,B 0,C 180,E1 -25962.295,E2 -25962.295} C_VEL
LIN {X 0,Y 147.121,Z 513.975,A -85,B 0,C 180,E1 -25964.246,E2 -25964.246} C_VEL
LIN {X 0,Y 140.445,Z 521.543,A -85,B 0,C 180,E1 -25967.519,E2 -25967.519} C_VEL
LIN {X 0,Y 134.169,Z 527.707,A -85,B 0,C 180,E1 -25971.07,E2 -25971.07} C_VEL
LIN {X 0,Y 128.769,Z 532.587,A -85,B 0,C 180,E1 -25974.953,E2 -25974.953} C_VEL
LIN {X 0,Y 123.79,Z 536.561,A -85,B 0,C 180,E1 -25979.287,E2 -25979.287} C_VEL
LIN {X 0,Y 118.477,Z 540.242,A -85,B 0,C 180,E1 -25985.48,E2 -25985.48} C_VEL
LIN {X 0,Y 116.36,Z 541.499,A -85,B 0,C 180,E1 -25988.766,E2 -25988.766} C_VEL
LIN {X 0,Y 113.601,Z 542.807,A -85,B 0,C 180,E1 -25995.685,E2 -25995.685} C_VEL
LIN {X 0,Y 112.36,Z 542.623,A -85,B 0,C 180,E1 -26002.826,E2 -26002.826} C_VEL
LIN {X 0,Y 112.26,Z 541.959,A -85,B 0,C 180,E1 -26006.423,E2 -26006.423} C_VEL
LIN {X 0,Y 112.448,Z 540.86,A -85,B 0,C 180,E1 -26010.012,E2 -26010.012} C_VEL
LIN {X 0,Y 112.34,Z 539.303,A -85,B 0,C 180,E1 -26013.598,E2 -26013.598} C_VEL
LIN {X 0,Y 112.62,Z 536.115,A -85,B 0,C 180,E1 -26018.987,E2 -26018.987} C_VEL
LIN {X 0,Y 113.577,Z 531.807,A -85,B 0,C 180,E1 -26024.341,E2 -26024.341} C_VEL
LIN {X 0,Y 115.358,Z 526.264,A -85,B 0,C 180,E1 -26029.588,E2 -26029.588} C_VEL
LIN {X 0,Y 118.016,Z 519.31,A -85,B 0,C 180,E1 -26034.647,E2 -26034.647} C_VEL
LIN {X 0,Y 120.881,Z 511.992,A -85,B 0,C 180,E1 -26038.786,E2 -26038.786} C_VEL
LIN {X 0,Y 124.275,Z 503.563,A -85,B 0,C 180,E1 -26042.506,E2 -26042.506} C_VEL
LIN {X 0,Y 127.136,Z 496.088,A -85,B 0,C 180,E1 -26045.137,E2 -26045.137} C_VEL
LIN {X 0,Y 128.174,Z 491.408,A -85,B 0,C 180,E1 -26046.704,E2 -26046.704} C_VEL
LIN {X 0,Y 128.27,Z 483.443,A -85,B 0,C 180,E1 -26049.37,E2 -26049.37} C_VEL
LIN {X 0,Y 128.36,Z 475.064,A -85,B 0,C 180,E1 -26051.754,E2 -26051.754} C_VEL
LIN {X 0,Y 129.324,Z 469.742,A -85,B 0,C 180,E1 -26052.819,E2 -26052.819} C_VEL
LIN {X 0,Y 132.526,Z 456.488,A -85,B 0,C 180,E1 -26054.651,E2 -26054.651} C_VEL
LIN {X 0,Y 134.657,Z 443.722,A -85,B 0,C 180,E1 -26055.87,E2 -26055.87} C_VEL
LIN {X 0,Y 136.064,Z 429.692,A -85,B 0,C 180,E1 -26056.691,E2 -26056.691} C_VEL
LIN {X 0,Y 138.382,Z 400.784,A -85,B 0,C 180,E1 -26058.069,E2 -26058.069} C_VEL
LIN {X 0,Y 138.011,Z 395.943,A -85,B 0,C 180,E1 -26058.547,E2 -26058.547} C_VEL
LIN {X 0,Y 132.932,Z 380.99,A -85,B 0,C 180,E1 -26061.489,E2 -26061.489} C_VEL
LIN {X 0,Y 128.292,Z 369.574,A -85,B 0,C 180,E1 -26064.252,E2 -26064.252} C_VEL
LIN {X 0,Y 125.022,Z 362.939,A -85,B 0,C 180,E1 -26066.281,E2 -26066.281} C_VEL
LIN {X 0,Y 119.865,Z 354.635,A -85,B 0,C 180,E1 -26069.622,E2 -26069.622} C_VEL
LIN {X 0,Y 116.98,Z 350.445,A -85,B 0,C 180,E1 -26071.641,E2 -26071.641} C_VEL
LIN {X 0,Y 114.58,Z 346.91,A -85,B 0,C 180,E1 -26073.474,E2 -26073.474} C_VEL
LIN {X 0,Y 112.283,Z 344.09,A -85,B 0,C 180,E1 -26075.307,E2 -26075.307} C_VEL
LIN {X 0,Y 111.284,Z 342.267,A -85,B 0,C 180,E1 -26076.201,E2 -26076.201} C_VEL
LIN {X 0,Y 109.019,Z 340.07,A -85,B 0,C 180,E1 -26078.118,E2 -26078.118} C_VEL
LIN {X 0,Y 108.046,Z 337.872,A -85,B 0,C 180,E1 -26079.162,E2 -26079.162} C_VEL
LIN {X 0,Y 107.893,Z 337.028,A -85,B 0,C 180,E1 -26079.505,E2 -26079.505} C_VEL
LIN {X 0,Y 108.152,Z 336.986,A -85,B 0,C 180,E1 -26087.132,E2 -26087.132} C_VEL
LIN {X 0,Y 108.303,Z 336.978,A -85,B 0,C 180,E1 -26092.543,E2 -26092.543} C_VEL
LIN {X 0,Y 108.916,Z 336.857,A -85,B 0,C 180,E1 -26100,E2 -26100} C_VEL
LIN {X 0,Y 108.299,Z 336.99,A -85,B 0,C 180,E1 -26107.458,E2 -26107.458} C_VEL
LIN {X 0,Y 108.151,Z 337.006,A -85,B 0,C 180,E1 -26112.867,E2 -26112.867} C_VEL
LIN {X 0,Y 107.868,Z 337.027,A -85,B 0,C 180,E1 -26119.012,E2 -26119.012} C_VEL
LIN {X 0,Y 107.802,Z 337.053,A -85,B 0,C 180,E1 -26124.097,E2 -26124.097} C_VEL
LIN {X 0,Y 107.76,Z 336.99,A -85,B 0,C 180,E1 -26132.006,E2 -26132.006} C_VEL
LIN {X 0,Y 107.688,Z 337.069,A -85,B 0,C 180,E1 -26138.435,E2 -26138.435} C_VEL
LIN {X 0,Y 107.676,Z 337.073,A -85,B 0,C 180,E1 -26145.887,E2 -26145.887} C_VEL
LIN {X 0,Y 107.728,Z 337.07,A -85,B 0,C 180,E1 -26153.132,E2 -26153.132} C_VEL
LIN {X 0,Y 108.602,Z 339.726,A -85,B 0,C 180,E1 -26154.182,E2 -26154.182} C_VEL
LIN {X 0,Y 110.62,Z 341.929,A -85,B 0,C 180,E1 -26155.959,E2 -26155.959} C_VEL
LIN {X 0,Y 111.621,Z 342.676,A -85,B 0,C 180,E1 -26156.749,E2 -26156.749} C_VEL
LIN {X 0,Y 113.54,Z 345.846,A -85,B 0,C 180,E1 -26158.405,E2 -26158.405} C_VEL
LIN {X 0,Y 115.228,Z 347.861,A -85,B 0,C 180,E1 -26159.708,E2 -26159.708} C_VEL
LIN {X 0,Y 121.28,Z 356.643,A -85,B 0,C 180,E1 -26163.989,E2 -26163.989} C_VEL
LIN {X 0,Y 127.63,Z 367.029,A -85,B 0,C 180,E1 -26167.917,E2 -26167.917} C_VEL
LIN {X 0,Y 133.082,Z 376.86,A -85,B 0,C 180,E1 -26170.918,E2 -26170.918} C_VEL
LIN {X 0,Y 139.073,Z 389.959,A -85,B 0,C 180,E1 -26174.023,E2 -26174.023} C_VEL
LIN {X 0,Y 135.388,Z 432.344,A -85,B 0,C 180,E1 -26176.08,E2 -26176.08} C_VEL
LIN {X 0,Y 133.432,Z 445.959,A -85,B 0,C 180,E1 -26177.303,E2 -26177.303} C_VEL
LIN {X 0,Y 130.86,Z 458.4,A -85,B 0,C 180,E1 -26178.96,E2 -26178.96} C_VEL
LIN {X 0,Y 127.679,Z 470.236,A -85,B 0,C 180,E1 -26181.132,E2 -26181.132} C_VEL
LIN {X 0,Y 123.975,Z 481.565,A -85,B 0,C 180,E1 -26183.888,E2 -26183.888} C_VEL
LIN {X 0,Y 120.174,Z 491.868,A -85,B 0,C 180,E1 -26187.218,E2 -26187.218} C_VEL
